// ---- POUs/HW/FB_EL2904_DiagnosticData.TcPOU
(****************************************************************************************)
(*							Beckhoff Automation Poland									*)
(*									30.01.2017											*)
(*			Blok funkcyjny pobierający informacje diagnostyczne z modułu EL2904			*)
(*			v2.5:																		*)
(*				- bReset, wErrorCount, ACT_Reset zmiana nazw pozostalych akcji			*)
(*				- usunieta zmienna sPath												*)
(*			v2.4:																		*)
(*				- obsluga bledu															*)
(*			v2.3:																		*)
(*				- dostosowano do rozbudowanej struktury									*)
(*			v1.2:																		*)
(*				- uruchamianie zboczem narastającym bExecute							*)	
(*______________________________________________________________________________________*)

FUNCTION_BLOCK FB_EL2904_DiagnosticData IMPLEMENTS I_ErrorHandling
VAR_INPUT
	sNetId						: T_AmsNetId;					(* Adres mastera EtherCAT *)
	uiSlaveAddr					: UINT;							(* Adres slave EtherCAT modułu EL2904 *)
	bExecute					: BOOL;							(* Zbocze narastające aktywuje komende *)
	bReset						: BOOL;							(* 	*)
END_VAR
VAR_OUTPUT
	stEL2904_DiagnosticData		: ST_EL2904_DiagnosticData;		(* Wyjściowa struktura danych *)
	bBusy						: BOOL;							(* Wyjście jest ustawione gdy aktualnie wykonywana jest komenda *)
	bError						: BOOL;							(* Wyjście jest ustawione gdy wystąpił błąd *) 
	udiErrorId					: UDINT;						(* Kod błedu *)
	bNewData					: BOOL;							(* Po otrzymaniu nowych danych przyjmuje wartość TRUE na jeden cykl *)
END_VAR
VAR
	fbEcCoESdoRead				: FB_EcCoESdoRead;
	stTempData					: ST_EL2904_DiagnosticData;		(* Tymczasowa struktura danych *)
	BSubIndex					: BYTE;
	wIndex						: WORD;
	iStep						: INT;
	pDstBuf						: PVOID;
	cbBufLen					: UDINT;
	rtExecute					: R_TRIG;
	rtError						: R_TRIG;
	rtReset						: R_TRIG;
	bRead						: BOOL;							(* Odczyt *)
	wTemp_800E_0C				: WORD;							(* Wartosc tymczasowa *)
	wTemp_800E_0D				: WORD;							(* Wartosc tymczasowa *)
	wTemp_800E_0E				: WORD;							(* Wartosc tymczasowa *)
	wErrorCount					: WORD;							// Licznik bledow
END_VAR

ACT_Reset(); 									// Wywolanie akcji resetu

rtExecute(CLK:=bExecute);

CASE iStep OF		
	(* Wspolne *)	
	0:												(* Odczyt nazwy modułu *)
		bNewData	:= FALSE;
		bRead		:= FALSE;
		IF rtExecute.Q THEN
			bBusy			:= TRUE;
			bError			:= FALSE;
			udiErrorId		:= 0;
			wIndex 			:= 16#1008;
			BSubIndex 		:= 0;
			pDstBuf 		:= ADR (stTempData.sDeviceName);
			cbBufLen 		:= SIZEOF(stTempData.sDeviceName);
			bRead			:= TRUE;
			iStep			:= iStep + 10;
		END_IF
	10:												(* Odczyt wersji HW *)
		bRead		:= FALSE;
		IF NOT fbEcCoESdoRead.bBusy AND NOT fbEcCoESdoRead.bError THEN
			wIndex 			:= 16#1009;
			BSubIndex 		:= 0;
			pDstBuf 		:= ADR (stTempData.sHardwareVersion);
			cbBufLen 		:= SIZEOF(stTempData.sHardwareVersion);
			bRead			:= TRUE;
			iStep			:= iStep + 10;
		END_IF
	20:												(* Odczyt wersji SW *)
		bRead				:= FALSE;
		IF NOT fbEcCoESdoRead.bBusy AND NOT fbEcCoESdoRead.bError THEN
			wIndex 			:= 16#100A;
			BSubIndex 		:= 0;
			pDstBuf 		:= ADR (stTempData.sSoftwareVersion);
			cbBufLen 		:= SIZEOF(stTempData.sSoftwareVersion);
			bRead			:= TRUE;
			iStep			:= iStep + 10;
		END_IF
	30:												(* Odczyt adresu FSoE *)
		bRead				:= FALSE;
		IF NOT fbEcCoESdoRead.bBusy AND NOT fbEcCoESdoRead.bError THEN
			wIndex 			:= 16#F980;
			BSubIndex 		:= 1;
			pDstBuf 		:= ADR (stTempData.dwFSoEAddress);
			cbBufLen 		:= SIZEOF(stTempData.dwFSoEAddress);
			bRead			:= TRUE;
			iStep			:= iStep + 10;
		END_IF;
	40:												(* Odczyt numeru seryjnego *)
		bRead				:= FALSE;
		IF NOT fbEcCoESdoRead.bBusy AND NOT fbEcCoESdoRead.bError THEN
			wIndex 			:= 16#F980;
			BSubIndex 		:= 2;
			pDstBuf 		:= ADR (stTempData.dwSerialNumber);
			cbBufLen 		:= SIZEOF(stTempData.dwSerialNumber);
			bRead			:= TRUE;
			iStep			:= iStep + 10;
		END_IF
	50:												(* Odczyt Temperature measurement 1 *)
		bRead				:= FALSE;
		IF NOT fbEcCoESdoRead.bBusy AND NOT fbEcCoESdoRead.bError THEN
			wIndex 			:= 16#FA80;
			BSubIndex 		:= 1;
			pDstBuf 		:= ADR (stTempData.wTemperaturePrimaryMC);
			cbBufLen 		:= SIZEOF(stTempData.wTemperaturePrimaryMC);
			bRead			:= TRUE;
			iStep			:= iStep + 10;
		END_IF
	60:												(* Odczyt Temperature measurement 2 *)
		bRead				:= FALSE;
		IF NOT fbEcCoESdoRead.bBusy AND NOT fbEcCoESdoRead.bError THEN
			wIndex 			:= 16#FA80;
			BSubIndex 		:= 2;
			pDstBuf 		:= ADR (stTempData.wTemperatureSecondaryMC);
			cbBufLen 		:= SIZEOF(stTempData.wTemperatureSecondaryMC);
			bRead			:= TRUE;
			iStep			:= iStep + 10;
		END_IF
	(*Charakterystyczne dla modulu *)
	70:												(* Odczyt FA80:03 Temperature Outputs *)
		bRead				:= FALSE;
		IF NOT fbEcCoESdoRead.bBusy AND NOT fbEcCoESdoRead.bError THEN
			wIndex 			:= 16#FA80;
			BSubIndex 		:= 3;
			pDstBuf 		:= ADR (stTempData.wTemperatureOut);
			cbBufLen 		:= SIZEOF(stTempData.wTemperatureOut);
			bRead			:= TRUE;
			iStep			:= iStep + 10;
		END_IF
	80:												(* Odczyt DO 1 *)
		bRead				:= FALSE;
		IF NOT fbEcCoESdoRead.bBusy AND NOT fbEcCoESdoRead.bError THEN
			wIndex 			:= 16#7001;
			BSubIndex 		:= 1;
			pDstBuf 		:= ADR(stTempData.bOutput1);
			cbBufLen 		:= SIZEOF(stTempData.bOutput1);
			bRead			:= TRUE;
			iStep			:= iStep + 10;
		END_IF
	90:												(* Odczyt DO 2 *)
		bRead				:= FALSE;
		IF NOT fbEcCoESdoRead.bBusy AND NOT fbEcCoESdoRead.bError THEN
			wIndex 			:= 16#7001;
			BSubIndex 		:= 2;
			pDstBuf 		:= ADR(stTempData.bOutput2);
			cbBufLen 		:= SIZEOF(stTempData.bOutput2);
			bRead			:= TRUE;
			iStep			:= iStep + 10;
		END_IF
	100:											(* Odczyt DO 3 *)
		bRead				:= FALSE;
		IF NOT fbEcCoESdoRead.bBusy AND NOT fbEcCoESdoRead.bError THEN
			wIndex 			:= 16#7001;
			BSubIndex 		:= 3;
			pDstBuf 		:= ADR(stTempData.bOutput3);
			cbBufLen 		:= SIZEOF(stTempData.bOutput3);
			bRead			:= TRUE;
			iStep			:= iStep + 10;
		END_IF
	110:											(* Odczyt DO 4 *)
		bRead				:= FALSE;
		IF NOT fbEcCoESdoRead.bBusy AND NOT fbEcCoESdoRead.bError THEN
			wIndex 			:= 16#7001;
			BSubIndex 		:= 4;
			pDstBuf 		:= ADR(stTempData.bOutput4);
			cbBufLen 		:= SIZEOF(stTempData.bOutput4);
			bRead			:= TRUE;
			iStep			:= iStep + 10;
		END_IF
	120:											(* Odczyt 800E 0C *)
		bRead				:= FALSE;
		IF NOT fbEcCoESdoRead.bBusy AND NOT fbEcCoESdoRead.bError THEN
			wIndex 			:= 16#800E;
			BSubIndex 		:= 16#0C;
			pDstBuf 		:= ADR (wTemp_800E_0C);
			cbBufLen 		:= SIZEOF(wTemp_800E_0C);
			bRead			:= TRUE;
			iStep			:= iStep + 10;
		END_IF
	130:											(* Odczyt 800E 0D *)
		bRead				:= FALSE;
		IF NOT fbEcCoESdoRead.bBusy AND NOT fbEcCoESdoRead.bError THEN
			wIndex 			:= 16#800E;
			BSubIndex 		:= 16#0D;
			pDstBuf 		:= ADR (wTemp_800E_0D);
			cbBufLen 		:= SIZEOF(wTemp_800E_0D);
			bRead			:= TRUE;
			iStep			:= iStep + 10;
		END_IF
	140:											(* Odczyt 800E 0E *)
		bRead				:= FALSE;
		IF NOT fbEcCoESdoRead.bBusy AND NOT fbEcCoESdoRead.bError THEN
			wIndex 			:= 16#800E;
			BSubIndex 		:= 16#0E;
			pDstBuf 		:= ADR (wTemp_800E_0E);
			cbBufLen 		:= SIZEOF(wTemp_800E_0E);
			bRead			:= TRUE;
			iStep			:= iStep + 10;
		END_IF
	
	150: (* Koniec odczytu *)
		bRead				:= FALSE;
		IF NOT fbEcCoESdoRead.bBusy AND NOT fbEcCoESdoRead.bError THEN
			iStep 			:= 200;
		END_IF
	200: (* Konwersje *)
		(* Zmiana numeru seryjnego na STRING *)
		stTempData.sSerialNumber 		:= '00000000';
		stTempData.sSerialNumber 		:= CONCAT(DELETE(stTempData.sSerialNumber, LEN(DWORD_TO_STRING(stTempData.dwSerialNumber)),1),DWORD_TO_STRING(stTempData.dwSerialNumber));
		stTempData.bOutputCross1 		:= wTemp_800E_0C.0;
		stTempData.bOutputCross2 		:= wTemp_800E_0C.1;
		stTempData.bOutputCross3 		:= wTemp_800E_0C.2;
		stTempData.bOutputCross4 		:= wTemp_800E_0C.3;
		stTempData.bOutputOpen1 		:= wTemp_800E_0C.4;
		stTempData.bOutputOpen2 		:= wTemp_800E_0C.5;
		stTempData.bOutputOpen3 		:= wTemp_800E_0C.6;
		stTempData.bOutputOpen4 		:= wTemp_800E_0C.7;
		stTempData.bFieldVoltH 			:= wTemp_800E_0D.0;
		stTempData.bFieldVoltL	 		:= wTemp_800E_0D.1;
		stTempData.bTHUC1			 	:= wTemp_800E_0E.0;
		stTempData.bTHUC2			 	:= wTemp_800E_0E.1;
		stTempData.bTOutBoardH		 	:= wTemp_800E_0E.2;
		stTempData.bTLUC1			 	:= wTemp_800E_0E.3;
		stTempData.bTLUC2			 	:= wTemp_800E_0E.4;
		stTempData.bTOutBoardL		 	:= wTemp_800E_0E.5;
		stTempData.bTDiffProcBoard	 	:= wTemp_800E_0E.6;
		stTempData.bTDiffBoards		 	:= wTemp_800E_0E.7;
		(* General Error bit *)
		stTempData.bGeneralError := stTempData.bOutputCross1 OR stTempData.bOutputCross2 OR stTempData.bOutputCross3 OR stTempData.bOutputCross4 OR
									stTempData.bOutputOpen1 OR stTempData.bOutputOpen2 OR stTempData.bOutputOpen3 OR stTempData.bOutputOpen4 OR
									stTempData.bFieldVoltH OR stTempData.bFieldVoltL OR stTempData.bTHUC1 OR stTempData.bTHUC2 OR stTempData.bTOutBoardH OR
									stTempData.bTLUC1 OR stTempData.bTLUC2 OR stTempData.bTOutBoardL OR stTempData.bTDiffProcBoard OR stTempData.bTDiffBoards;
		
		(* Przepisanie danych tymczasowych na wyjscie *)	
		stEL2904_DiagnosticData := stTempData;
		(* Ustawienie flag i powrot do poczatku *)
		bBusy							:= FALSE;
		bNewData						:= TRUE;
		iStep 							:= 0;
	1000: (* ERROR *)
		wErrorCount 					:= wErrorCount + 1;			// Inkrementacja licznika bledow
		iStep 							:= 0;
END_CASE

fbEcCoESdoRead(
	sNetId		:= sNetId,
	nSlaveAddr	:= uiSlaveAddr,
	nSubIndex	:= BSubIndex,
	nIndex		:= wIndex,
	pDstBuf		:= pDstBuf,
	cbBufLen	:= cbBufLen,
	bExecute 	:= bRead);
	
ACT_Error();

ACTION ACT_Error:
rtError(CLK:= fbEcCoESdoRead.bError, Q=> );
IF rtError.Q THEN
	bBusy 			:= FALSE;
	bError 			:= TRUE;
	bRead			:= FALSE;
	udiErrorId 		:= fbEcCoESdoRead.nErrId;
	iStep 			:= 1000;
END_IF
END_ACTION

ACTION ACT_Reset:
rtReset(CLK:= bReset, Q=> );			// Wywolanie triggera, wykrycie zbocza narastajacego zmiennej wejsciowej bReset
IF rtReset.Q THEN
	bBusy						:= FALSE;
	bError						:= FALSE;
	bNewData					:= FALSE;
	bRead						:= FALSE;
	iStep						:= 0;
	udiErrorId					:= 0;
END_IF
END_ACTION

PROPERTY P_Error : BOOL
GET
END_GET
END_PROPERTY

PROPERTY P_ErrorID : UDINT
GET
END_GET
END_PROPERTY

{attribute 'object_name' := 'ToString'}
METHOD ToString : STRING(255)
END_METHOD

END_FUNCTION_BLOCK

// ---- POUs/HW/FB_EL6900_DiagnosticData.TcPOU
(****************************************************************************************)
(*							Beckhoff Automation Poland									*)
(*									30.01.2017											*)
(*			Blok funkcyjny pobierający informacje diagnostyczne z modułu EL6900			*)
(*			v2.5:																		*)
(*				- bReset, wErrorCount, ACT_Reset zmiana nazw pozostalych akcji			*)
(*				- usunieta zmienna sPath												*)
(*			v2.4:																		*)
(*				- obsluga bledu															*)
(*			v2.3:																		*)
(*				- dostosowano do rozbudowanej struktury									*)
(*			v1.2:																		*)
(*				- uruchamianie zboczem narastającym bExecute							*)	
(*______________________________________________________________________________________*)

FUNCTION_BLOCK FB_EL6900_DiagnosticData IMPLEMENTS I_ErrorHandling
VAR_INPUT
	sNetId						: T_AmsNetId;					(* Adres mastera EtherCAT *)
	uiSlaveAddr					: UINT;							(* Adres slave EtherCAT modułu EL6900 *)
	bExecute					: BOOL;							(* Zbocze narastające aktywuje komende *)
	bReset						: BOOL;							(* 	*)
END_VAR
VAR_OUTPUT
	stEL6900_DiagnosticData		: ST_EL6900_DiagnosticData;		(* Wyjściowa struktura danych *)
	bBusy						: BOOL;							(* Wyjście jest ustawione gdy aktualnie wykonywana jest komenda *)
	bError						: BOOL;							(* Wyjście jest ustawione gdy wystąpił błąd *) 
	udiErrorId					: UDINT;						(* Kod błedu *)
	bNewData					: BOOL;							(* Po otrzymaniu nowych danych przyjmuje wartość TRUE na jeden cykl *)
END_VAR
VAR
	fbEcCoESdoRead				: FB_EcCoESdoRead;
	stTempData					: ST_EL6900_DiagnosticData;		(* Tymczasowa struktura danych *)
	BSubIndex					: BYTE;
	wIndex						: WORD;
	iStep						: INT;
	pDstBuf						: PVOID;
	cbBufLen					: UDINT;
	rtExecute					: R_TRIG;
	rtError						: R_TRIG;
	rtReset						: R_TRIG;
	bRead						: BOOL;							(* Odczyt *)
	wTemp_FA00_03				: WORD;							(* Wartosc tymczasowa *)
	wErrorCount					: WORD;							// Licznik bledow
END_VAR

ACT_Reset(); 									// Wywolanie akcji resetu

rtExecute(CLK:=bExecute);

CASE iStep OF		
	
	(* Wspolne *)	
	0:												(* Odczyt nazwy modułu *)
		bNewData	:= FALSE;
		bRead		:= FALSE;
		IF rtExecute.Q THEN
			bBusy			:= TRUE;
			bError			:= FALSE;
			udiErrorId		:= 0;
			wIndex 			:= 16#1008;
			BSubIndex 		:= 0;
			pDstBuf 		:= ADR (stTempData.sDeviceName);
			cbBufLen 		:= SIZEOF(stTempData.sDeviceName);
			bRead			:= TRUE;
			iStep			:= iStep + 10;
		END_IF
	10:												(* Odczyt wersji HW *)
		bRead		:= FALSE;
		IF NOT fbEcCoESdoRead.bBusy AND NOT fbEcCoESdoRead.bError THEN
			wIndex 			:= 16#1009;
			BSubIndex 		:= 0;
			pDstBuf 		:= ADR (stTempData.sHardwareVersion);
			cbBufLen 		:= SIZEOF(stTempData.sHardwareVersion);
			bRead			:= TRUE;
			iStep			:= iStep + 10;
		END_IF
	20:												(* Odczyt wersji SW *)
		bRead				:= FALSE;
		IF NOT fbEcCoESdoRead.bBusy AND NOT fbEcCoESdoRead.bError THEN
			wIndex 			:= 16#100A;
			BSubIndex 		:= 0;
			pDstBuf 		:= ADR (stTempData.sSoftwareVersion);
			cbBufLen 		:= SIZEOF(stTempData.sSoftwareVersion);
			bRead			:= TRUE;
			iStep			:= iStep + 10;
		END_IF
	30:												(* Odczyt adresu FSoE *)
		bRead				:= FALSE;
		IF NOT fbEcCoESdoRead.bBusy AND NOT fbEcCoESdoRead.bError THEN
			wIndex 			:= 16#F980;
			BSubIndex 		:= 1;
			pDstBuf 		:= ADR (stTempData.dwFSoEAddress);
			cbBufLen 		:= SIZEOF(stTempData.dwFSoEAddress);
			bRead			:= TRUE;
			iStep			:= iStep + 10;
		END_IF;
	40:												(* Odczyt numeru seryjnego *)
		bRead				:= FALSE;
		IF NOT fbEcCoESdoRead.bBusy AND NOT fbEcCoESdoRead.bError THEN
			wIndex 			:= 16#F980;
			BSubIndex 		:= 2;
			pDstBuf 		:= ADR (stTempData.dwSerialNumber);
			cbBufLen 		:= SIZEOF(stTempData.dwSerialNumber);
			bRead			:= TRUE;
			iStep			:= iStep + 10;
		END_IF
	50:												(* Odczyt Temperature measurement 1 *)
		bRead				:= FALSE;
		IF NOT fbEcCoESdoRead.bBusy AND NOT fbEcCoESdoRead.bError THEN
			wIndex 			:= 16#FA80;
			BSubIndex 		:= 1;
			pDstBuf 		:= ADR (stTempData.wTemperaturePrimaryMC);
			cbBufLen 		:= SIZEOF(stTempData.wTemperaturePrimaryMC);
			bRead			:= TRUE;
			iStep			:= iStep + 10;
		END_IF
	60:												(* Odczyt Temperature measurement 2 *)
		bRead				:= FALSE;
		IF NOT fbEcCoESdoRead.bBusy AND NOT fbEcCoESdoRead.bError THEN
			wIndex 			:= 16#FA80;
			BSubIndex 		:= 2;
			pDstBuf 		:= ADR (stTempData.wTemperatureSecondaryMC);
			cbBufLen 		:= SIZEOF(stTempData.wTemperatureSecondaryMC);
			bRead			:= TRUE;
			iStep			:= iStep + 10;
		END_IF
	(*Charakterystyczne dla modulu *)
	70:												(* Odczyt CRC projektu *)
		bRead				:= FALSE;
		IF NOT fbEcCoESdoRead.bBusy AND NOT fbEcCoESdoRead.bError THEN
			wIndex 			:= 16#F980;
			BSubIndex 		:= 3;
			pDstBuf 		:= ADR (stTempData.dwProjectCRC);
			cbBufLen 		:= SIZEOF(stTempData.dwProjectCRC);
			bRead			:= TRUE;
			iStep			:= iStep + 10;
		END_IF
	80:												(* Odczyt Safety Project State *)
		bRead				:= FALSE;
		IF NOT fbEcCoESdoRead.bBusy AND NOT fbEcCoESdoRead.bError THEN
			wIndex 			:= 16#F100;
			BSubIndex 		:= 1;
			pDstBuf 		:= ADR (stTempData.wSafetyProjectState);
			cbBufLen 		:= SIZEOF(stTempData.wSafetyProjectState);
			bRead			:= TRUE;
			iStep			:= iStep + 10;
		END_IF
	90:												(* Odczyt Vcc Primary MC*)
		bRead				:= FALSE;
		IF NOT fbEcCoESdoRead.bBusy AND NOT fbEcCoESdoRead.bError THEN
			wIndex 			:= 16#FA80;
			BSubIndex 		:= 3;
			pDstBuf 		:= ADR (stTempData.wVccPrimaryMC);
			cbBufLen 		:= SIZEOF(stTempData.wVccPrimaryMC);
			bRead			:= TRUE;
			iStep			:= iStep + 10;
		END_IF
	100:											(* Odczyt Vcc Secondary MC*)
		bRead				:= FALSE;
		IF NOT fbEcCoESdoRead.bBusy AND NOT fbEcCoESdoRead.bError THEN
			wIndex 			:= 16#FA80;
			BSubIndex 		:= 4;
			pDstBuf 		:= ADR (stTempData.wVccSecondaryMC);
			cbBufLen 		:= SIZEOF(stTempData.wVccSecondaryMC);
			bRead			:= TRUE;
			iStep			:= iStep + 10;
		END_IF
	110:											(* Odczyt FA00:03 Temperature error / Supply error *)
		bRead				:= FALSE;
		IF NOT fbEcCoESdoRead.bBusy AND NOT fbEcCoESdoRead.bError THEN
			wIndex 			:= 16#FA00;
			BSubIndex 		:= 3;
			pDstBuf 		:= ADR (wTemp_FA00_03);
			cbBufLen 		:= SIZEOF(wTemp_FA00_03);
			bRead			:= TRUE;
			iStep			:= iStep + 10;
		END_IF
	120: (* Koniec odczytu *)
		bRead				:= FALSE;
		IF NOT fbEcCoESdoRead.bBusy AND NOT fbEcCoESdoRead.bError THEN
			iStep 			:= 200;
		END_IF
	200: (* Konwersje *)
		(* Zmiana numeru seryjnego na STRING *)
		stTempData.sSerialNumber 		:= '00000000';
		stTempData.sSerialNumber 		:= CONCAT(DELETE(stTempData.sSerialNumber, LEN(DWORD_TO_STRING(stTempData.dwSerialNumber)),1),DWORD_TO_STRING(stTempData.dwSerialNumber));
		(* Zmiana CRC na STRING *)
		stTempData.sProjectCRC 			:= F_SAFETY_DWORD_TO_STIRNGHEX(stTempData.dwProjectCRC);
		(* Zmiana Project State na ENUM *)
		stTempData.eSAFETY_ProjectState	:= WORD_TO_INT(stTempData.wSafetyProjectState);
		(* Dekodowanie FA00:03 Temperature error / Supply error *)
		stTempData.bTempMax 			:= wTemp_FA00_03 = 16#0005;
		stTempData.bTempMin 			:= wTemp_FA00_03 = 16#0006;
		stTempData.bTempDiff 			:= wTemp_FA00_03 = 16#0007;
		stTempData.bSuppVoltuMaxC1		:= wTemp_FA00_03 = 16#0101;
		stTempData.bSuppVoltuMaxC2		:= wTemp_FA00_03 = 16#0102;
		stTempData.bSuppVoltuMinC1		:= wTemp_FA00_03 = 16#0103;
		stTempData.bSuppVoltuMinC2		:= wTemp_FA00_03 = 16#0104;
		(* General Error bit *)
		stTempData.bGeneralError := stTempData.bTempMax OR stTempData.bTempMin OR stTempData.bTempDiff OR
									stTempData.bSuppVoltuMaxC1 OR stTempData.bSuppVoltuMaxC2 OR stTempData.bSuppVoltuMinC1 OR stTempData.bSuppVoltuMinC2;
		(* Przepisanie danych tymczasowych na wyjscie *)	
		stEL6900_DiagnosticData 		:= stTempData;
		(* Ustawienie flag i powrot do poczatku *)
		bBusy							:= FALSE;
		bNewData						:= TRUE;
		iStep 							:= 0;
	1000: (* ERROR *)
		wErrorCount 					:= wErrorCount + 1;			// Inkrementacja licznika bledow
		iStep 							:= 0;
END_CASE

fbEcCoESdoRead(
	sNetId		:= sNetId,
	nSlaveAddr	:= uiSlaveAddr,
	nSubIndex	:= BSubIndex,
	nIndex		:= wIndex,
	pDstBuf		:= pDstBuf,
	cbBufLen	:= cbBufLen,
	bExecute 	:= bRead);
	
ACT_Error();

ACTION ACT_Error:
rtError(CLK:= fbEcCoESdoRead.bError, Q=> );
IF rtError.Q THEN
	bBusy 			:= FALSE;
	bError 			:= TRUE;
	bRead			:= FALSE;
	udiErrorId 		:= fbEcCoESdoRead.nErrId;
	iStep 			:= 1000;
END_IF
END_ACTION

ACTION ACT_Reset:
rtReset(CLK:= bReset, Q=> );			// Wywolanie triggera, wykrycie zbocza narastajacego zmiennej wejsciowej bReset
IF rtReset.Q THEN
	bBusy						:= FALSE;
	bError						:= FALSE;
	bNewData					:= FALSE;
	bRead						:= FALSE;
	iStep						:= 0;
	udiErrorId					:= 0;
END_IF
END_ACTION

PROPERTY P_Error : BOOL
GET
END_GET
END_PROPERTY

PROPERTY P_ErrorID : UDINT
GET
END_GET
END_PROPERTY

{attribute 'object_name' := 'ToString'}
METHOD ToString : STRING(255)
END_METHOD

END_FUNCTION_BLOCK

// ---- POUs/Others/F_SAFETY_DWORD_TO_STIRNGHEX.TcPOU
///*************************************************************************************************************************
///							Beckhoff Automation Poland									
///				`        	F_SAFETY_DWORD_TO_STIRNGHEX v1.0							
///									13.03.2015											
///				Funkcja zwraca napis zawierający zapis liczby w formacie szesnastkowym.			
///_______________________________________________________________________________________
FUNCTION F_SAFETY_DWORD_TO_STIRNGHEX : STRING(8)
VAR_INPUT
	dwIn: DWORD;
END_VAR
VAR
	dwTemp: DWORD;
	i: INT;
END_VAR

FOR i := 0 TO 7 DO
	dwTemp := ROR(dwIn,4*i) AND 16#F;

	CASE dwTemp OF
	0..9:
		F_SAFETY_DWORD_TO_STIRNGHEX := CONCAT(DWORD_TO_STRING(dwTemp), F_SAFETY_DWORD_TO_STIRNGHEX);
	10:
		F_SAFETY_DWORD_TO_STIRNGHEX := CONCAT('A', F_SAFETY_DWORD_TO_STIRNGHEX);
	11:
		F_SAFETY_DWORD_TO_STIRNGHEX := CONCAT('B', F_SAFETY_DWORD_TO_STIRNGHEX);
	12:
		F_SAFETY_DWORD_TO_STIRNGHEX := CONCAT('C', F_SAFETY_DWORD_TO_STIRNGHEX);
	13:
		F_SAFETY_DWORD_TO_STIRNGHEX := CONCAT('D', F_SAFETY_DWORD_TO_STIRNGHEX);
	14:
		F_SAFETY_DWORD_TO_STIRNGHEX := CONCAT('E', F_SAFETY_DWORD_TO_STIRNGHEX);
	15:
		F_SAFETY_DWORD_TO_STIRNGHEX := CONCAT('F', F_SAFETY_DWORD_TO_STIRNGHEX);
	END_CASE;
END_FOR
F_SAFETY_DWORD_TO_STIRNGHEX := DELETE(F_SAFETY_DWORD_TO_STIRNGHEX,4,1);

END_FUNCTION

// ---- POUs/HW/FB_EL6900_StatusData.TcPOU
(****************************************************************************************)
(*							Beckhoff Automation Poland									*)
(*									03.03.2017											*)
(*				Blok funkcyjny pobierający informacje diagnostyczne						*)
(*			 o blokach funkcyjnych, grupach, polaczeniach z modułu EL6900				*)
(*			V2.6:																		*)
(*				- Poprawiono bugi pętli FOR odczytu w akcjach ACT_StatusConnections		*)
(*					ACT_StatusFunctionBlocks i ACT_StatusGroups							*)
(*			v2.5:																		*)
(*				- bReset, wErrorCount, ACT_Reset zmiana nazw pozostalych akcji			*)
(*				- usunieta zmienna sPath												*)
(*			v2.4:																		*)
(*				- obsluga bledu															*)
(*			v2.3:																		*)
(*				- dostosowano do rozbudowanej struktury									*)
(*			v1.2:																		*)
(*				- uruchamianie zboczem narastającym bExecute							*)	
(*______________________________________________________________________________________*)

FUNCTION_BLOCK FB_EL6900_StatusData IMPLEMENTS I_ErrorHandling
VAR_INPUT
	sNetId						: T_AmsNetId;					(* Adres mastera EtherCAT *)
	uiSlaveAddr					: UINT;							(* Adres slave EtherCAT modułu EL6900 *)
	bExecute					: BOOL;							(* Zbocze narastające aktywuje komende *)
	bReset						: BOOL;							(* 	*)
END_VAR
VAR_OUTPUT
	stEL6900_StatusData			: ST_EL6900_StatusData;			(* Wyjściowa struktura danych *)
	bBusy						: BOOL;							(* Wyjście jest ustawione gdy aktualnie wykonywana jest komenda *)
	bError						: BOOL;							(* Wyjście jest ustawione gdy wystąpił błąd *) 
	udiErrorId					: UDINT;						(* Kod błedu *)
	bNewData					: BOOL;							(* Po otrzymaniu nowych danych przyjmuje wartość TRUE na jeden cykl *)
END_VAR
VAR
	fbEcCoESdoRead				: FB_EcCoESdoRead;
	BSubIndex					: BYTE;
	wIndex						: WORD;
	iInit						: INT:=10;
	pDstBuf						: PVOID;
	cbBufLen					: UDINT;
	ftRead						: F_TRIG;
	udiLastErrorID				: UDINT;
	tonRead						: TON;
	iStep						: INT:=0;
	BStatusConnections			: BYTE:=0;
	dwTempStatusConnection		: DWORD;						(* Wartosc tymczasowa *)
	BStatusGroups				: BYTE:=0;
	dwTempStatusGroups			: DWORD;						(* Wartosc tymczasowa *)
	BStatusFunctionBlocks		: BYTE:= 0;
	stEL6900_StatusData_Temp	: ST_EL6900_StatusData;			(* Wartosc tymczasowa *)
	index						: INT;
	bRead						: BOOL;
	rtExecute					: R_TRIG;
	rtError						: R_TRIG;
	rtReset						: R_TRIG;
	wErrorCount					: WORD;							// Licznik bledow
END_VAR

ACT_Reset(); 									// Wywolanie akcji resetu

rtExecute(CLK:=bExecute);
CASE iStep OF
	0:
		ACT_Init();
	10:
		bNewData:=FALSE;
		IF rtExecute.Q THEN
			iStep:=20;
			bBusy:=TRUE;
			bError:=FALSE;
			udiErrorId:=0;
		END_IF
	20:
		ACT_StatusConnections();

	30:
		ACT_StatusGroups();

	40:
		ACT_StatusFunctionBlocks();
	50:
		stEL6900_StatusData := stEL6900_StatusData_Temp;
		iStep:=10;
		bBusy:=FALSE;
		bNewData:=TRUE;
		bRead:=FALSE;
	1000:
		wErrorCount 					:= wErrorCount + 1;			// Inkrementacja licznika bledow
		iStep 							:= 0;
END_CASE

fbEcCoESdoRead(
	sNetId		:= sNetId,
	nSlaveAddr	:= uiSlaveAddr,
	nSubIndex	:= BSubIndex,
	nIndex		:= wIndex,
	pDstBuf		:= pDstBuf,
	cbBufLen	:= cbBufLen,
	bExecute 	:= bRead);
	
ACT_Error();

ACTION ACT_Error:
rtError(CLK:= fbEcCoESdoRead.bError, Q=> );
IF rtError.Q THEN
	bBusy 			:= FALSE;
	bError 			:= TRUE;
	bRead			:= FALSE;
	udiErrorId 		:= fbEcCoESdoRead.nErrId;
	iStep 			:= 1000;
END_IF
END_ACTION

ACTION ACT_Init:
CASE iInit OF
10:
	bRead:=FALSE;
	IF rtExecute.Q THEN
		bBusy:=TRUE;
		bError:=FALSE;
		udiErrorId:=0;
		bNewData:=FALSE;
		wIndex 			:= 16#2110;
		BSubIndex 		:= 0;
		pDstBuf 		:= ADR(stEL6900_StatusData_Temp.dwStatusConnections);
		cbBufLen 		:= SIZEOF(stEL6900_StatusData_Temp.dwStatusConnections);
		iInit:=iInit+10;
		bRead:=TRUE;
	END_IF
20:
	bRead:=FALSE;
	IF NOT fbEcCoESdoRead.bError AND NOT fbEcCoESdoRead.bBusy THEN
		wIndex 			:= 16#2120;
		BSubIndex 		:= 0;
		pDstBuf 		:= ADR(stEL6900_StatusData_Temp.dwStatusGroups);
		cbBufLen 		:= SIZEOF(stEL6900_StatusData_Temp.dwStatusGroups);
		iInit:=iInit+10;
		bRead:=TRUE;
	END_IF
30:
	bRead:=FALSE;
	IF NOT fbEcCoESdoRead.bError AND NOT fbEcCoESdoRead.bBusy THEN
		wIndex 			:= 16#2130;
		BSubIndex 		:= 0;
		pDstBuf 		:= ADR(stEL6900_StatusData_Temp.dwStatusFunctionBlocks);
		cbBufLen 		:= SIZEOF(stEL6900_StatusData_Temp.dwStatusFunctionBlocks);
		iInit:=iInit+10;
		bRead:=TRUE;
	END_IF
ELSE
	bRead:=FALSE;
	iInit:=10;
	iStep:=20;
END_CASE
END_ACTION

ACTION ACT_Reset:
rtReset(CLK:= bReset, Q=> );			// Wywolanie triggera, wykrycie zbocza narastajacego zmiennej wejsciowej bReset
IF rtReset.Q THEN
	bBusy						:= FALSE;
	bError						:= FALSE;
	bNewData					:= FALSE;
	bRead						:= FALSE;
	iStep						:= 0;
	udiErrorId					:= 0;
END_IF
END_ACTION

ACTION ACT_StatusConnections:
bRead:=FALSE;
IF NOT fbEcCoESdoRead.bError AND NOT fbEcCoESdoRead.bBusy THEN
	BStatusConnections := BStatusConnections + 1;
	IF bStatusConnections>1 THEN
		stEL6900_StatusData_Temp.arrstStatusConnections[BStatusConnections-1].dwStatusConnection := (dwTempStatusConnection);
		stEL6900_StatusData_Temp.arrstStatusConnections[BStatusConnections-1].BState:= DWORD_TO_BYTE(dwTempStatusConnection AND 16#000000FF);(*1B*)
		stEL6900_StatusData_Temp.arrstStatusConnections[BStatusConnections-1].BDiagnosis := DWORD_TO_BYTE(ROR(dwTempStatusConnection AND 16#0000FF00,8));(*2B*)
		stEL6900_StatusData_Temp.arrstStatusConnections[BStatusConnections-1].eSAFETY_ConnectionState:= stEL6900_StatusData_Temp.arrstStatusConnections[BStatusConnections-1].BState;
		stEL6900_StatusData_Temp.arrstStatusConnections[BStatusConnections-1].eSAFETY_ConnectionDiag0F := stEL6900_StatusData_Temp.arrstStatusConnections[BStatusConnections-1].BDiagnosis AND 16#0F;
		stEL6900_StatusData_Temp.arrstStatusConnections[BStatusConnections-1].BSAFETY_ConnectionDiagF0 := stEL6900_StatusData_Temp.arrstStatusConnections[BStatusConnections-1].BDiagnosis AND 16#F0;
		stEL6900_StatusData_Temp.arrstStatusConnections[BStatusConnections-1].sSAFETY_ConnectionDiagF0 := BYTE_TO_BINSTR(SHR(stEL6900_StatusData_Temp.arrstStatusConnections[BStatusConnections-1].BDiagnosis,4),4);
	END_IF
	IF BStatusConnections > stEL6900_StatusData_Temp.dwStatusConnections THEN
		BStatusConnections := 0;
		iStep := iStep + 10;
		bRead:=FALSE;
	ELSE
		wIndex 			:= 16#2110;
		BSubIndex 		:= 0+BStatusConnections;
		pDstBuf 		:= ADR(dwTempStatusConnection);
		cbBufLen 		:= SIZEOF(dwTempStatusConnection);
		bRead:=TRUE;
	END_IF
END_IF
END_ACTION

ACTION ACT_StatusFunctionBlocks:
bRead:=FALSE;
IF NOT fbEcCoESdoRead.bError AND NOT fbEcCoESdoRead.bBusy THEN
	BStatusFunctionBlocks := BStatusFunctionBlocks + 1;
	IF BStatusFunctionBlocks > stEL6900_StatusData_Temp.dwStatusFunctionBlocks THEN
		bRead:=FALSE;
		BStatusFunctionBlocks := 0;
		iStep := 50;
	ELSE
		wIndex 			:= 16#2130;
		BSubIndex 		:= BStatusFunctionBlocks;
		pDstBuf 		:= ADR(stEL6900_StatusData_Temp.arrstStatusFunctionBlocks[BStatusFunctionBlocks]);
		cbBufLen 		:= SIZEOF(stEL6900_StatusData_Temp.arrstStatusFunctionBlocks[BStatusFunctionBlocks]);
		bRead:=TRUE;
	END_IF
END_IF
END_ACTION

ACTION ACT_StatusGroups:
bRead:=FALSE;
IF NOT fbEcCoESdoRead.bError AND NOT fbEcCoESdoRead.bBusy THEN
	BStatusGroups := BStatusGroups + 1;	
	IF BStatusGroups>1 THEN
		stEL6900_StatusData_Temp.arrstStatusGroups[BStatusGroups-1].dwStatusGroup := dwTempStatusGroups;
		stEL6900_StatusData_Temp.arrstStatusGroups[BStatusGroups-1].BState := DWORD_TO_BYTE(dwTempStatusGroups AND 16#000000FF);
		stEL6900_StatusData_Temp.arrstStatusGroups[BStatusGroups-1].eSAFETY_GroupState := stEL6900_StatusData_Temp.arrstStatusGroups[BStatusGroups-1].BState;
		stEL6900_StatusData_Temp.arrstStatusGroups[BStatusGroups-1].BDiagnosis := DWORD_TO_BYTE(ROR(dwTempStatusGroups AND 16#0000FF00,8));(*2B*)
		stEL6900_StatusData_Temp.arrstStatusGroups[BStatusGroups-1].BInputs := DWORD_TO_BYTE(ROR(dwTempStatusGroups AND 16#00FF0000,16));(*3B*)
		stEL6900_StatusData_Temp.arrstStatusGroups[BStatusGroups-1].BOutputs := DWORD_TO_BYTE(ROR(dwTempStatusGroups AND 16#FF000000,24));(*4B*)
		stEL6900_StatusData_Temp.arrstStatusGroups[BStatusGroups-1].bRUN_STOP := stEL6900_StatusData_Temp.arrstStatusGroups[BStatusGroups-1].BInputs.0;
		stEL6900_StatusData_Temp.arrstStatusGroups[BStatusGroups-1].bERR_Ack := stEL6900_StatusData_Temp.arrstStatusGroups[BStatusGroups-1].BInputs.1;
		stEL6900_StatusData_Temp.arrstStatusGroups[BStatusGroups-1].bFB_ERR := stEL6900_StatusData_Temp.arrstStatusGroups[BStatusGroups-1].BOutputs.0;
		stEL6900_StatusData_Temp.arrstStatusGroups[BStatusGroups-1].bCOM_ERR := stEL6900_StatusData_Temp.arrstStatusGroups[BStatusGroups-1].BOutputs.1;
		stEL6900_StatusData_Temp.arrstStatusGroups[BStatusGroups-1].bOUT_ERR := stEL6900_StatusData_Temp.arrstStatusGroups[BStatusGroups-1].BOutputs.2;
	END_IF
	IF BStatusGroups > stEL6900_StatusData_Temp.dwStatusGroups THEN
		BStatusGroups := 0;
		iStep := iStep + 10;
		bRead:=FALSE;
	ELSE
		wIndex 			:= 16#2120;
		BSubIndex 		:= BStatusGroups;
		pDstBuf 		:= ADR(dwTempStatusGroups);
		cbBufLen 		:= SIZEOF(dwTempStatusGroups);
		bRead:=TRUE;
	END_IF
END_IF
END_ACTION

PROPERTY P_Error : BOOL
GET
END_GET
END_PROPERTY

PROPERTY P_ErrorID : UDINT
GET
END_GET
END_PROPERTY

{attribute 'object_name' := 'ToString'}
METHOD ToString : STRING(255)
END_METHOD

END_FUNCTION_BLOCK

// ---- POUs/FBs/F_SAFETY_StatusFB_TO_AND.TcPOU
FUNCTION F_SAFETY_StatusFB_TO_AND 	: ST_SAFETY_FBAND 		(* Struktura dedykowana *)
VAR_INPUT
	stFBStatus						: ST_SAFETY_FBStatus; 	(* Struktura ogolna *)
END_VAR

F_SAFETY_StatusFB_TO_AND.uStatus.stStatusWords 		:= stFBStatus;									(* Przepisanie *)
F_SAFETY_StatusFB_TO_AND.eState					 	:= stFBStatus.BState;							(* Ustawienie enum *)

END_FUNCTION

// ---- POUs/FBs/F_SAFETY_StatusFB_TO_CONNECTIONSHUTDOWN.TcPOU
FUNCTION F_SAFETY_StatusFB_TO_CONNECTIONSHUTDOWN : ST_SAFETY_FBCONNECTIONSHUTDOWN
VAR_INPUT
	stFBStatus						: ST_SAFETY_FBStatus; 	(* Struktura ogolna *)
END_VAR

F_SAFETY_StatusFB_TO_CONNECTIONSHUTDOWN.uStatus.stStatusWords	:= stFBStatus;									(* Przepisanie *)
F_SAFETY_StatusFB_TO_CONNECTIONSHUTDOWN.eState 					:= stFBStatus.BState;							(* Ustawienie enum *)
F_SAFETY_StatusFB_TO_CONNECTIONSHUTDOWN.bGeneralError			:= stFBStatus.wDiagnosis <> 0;					(* General Error *)

END_FUNCTION

// ---- POUs/FBs/F_SAFETY_StatusFB_TO_DECOUPLE.TcPOU
FUNCTION F_SAFETY_StatusFB_TO_DECOUPLE : ST_SAFETY_FBDECOUPLE
VAR_INPUT
	stFBStatus						: ST_SAFETY_FBStatus; 	(* Struktura ogolna *)
END_VAR

F_SAFETY_StatusFB_TO_DECOUPLE.uStatus.stStatusWords 		:= stFBStatus;					(* Przepisanie *)
F_SAFETY_StatusFB_TO_DECOUPLE.eState					 	:= stFBStatus.BState;			(* Ustawienie enum *)

END_FUNCTION

// ---- POUs/FBs/F_SAFETY_StatusFB_TO_EDM.TcPOU
FUNCTION F_SAFETY_StatusFB_TO_EDM : ST_SAFETY_FBEDM
VAR_INPUT
	stFBStatus						: ST_SAFETY_FBStatus; 	(* Struktura ogolna *)
END_VAR

F_SAFETY_StatusFB_TO_EDM.uStatus.stStatusWords	:= stFBStatus;									(* Przepisanie *)
F_SAFETY_StatusFB_TO_EDM.eState 				:= stFBStatus.BState;							(* Ustawienie enum *)
F_SAFETY_StatusFB_TO_EDM.bGeneralError			:= stFBStatus.wDiagnosis <> 0;					(* General Error *)

END_FUNCTION

// ---- POUs/FBs/F_SAFETY_StatusFB_TO_ESTOP.TcPOU
FUNCTION F_SAFETY_StatusFB_TO_ESTOP : ST_SAFETY_FBESTOP 	(* Struktura dedykowana *)
VAR_INPUT
	stFBStatus						: ST_SAFETY_FBStatus; 	(* Struktura ogolna *)
END_VAR

F_SAFETY_StatusFB_TO_ESTOP.uStatus.stStatusWords	:= stFBStatus;									(* Przepisanie *)
F_SAFETY_StatusFB_TO_ESTOP.eState 					:= stFBStatus.BState;							(* Ustawienie enum *)
F_SAFETY_StatusFB_TO_ESTOP.bGeneralError			:= stFBStatus.wDiagnosis <> 0;					(* General Error *)

END_FUNCTION

// ---- POUs/FBs/F_SAFETY_StatusFB_TO_MON.TcPOU
FUNCTION F_SAFETY_StatusFB_TO_MON : ST_SAFETY_FBMON
VAR_INPUT
	stFBStatus						: ST_SAFETY_FBStatus; 	(* Struktura ogolna *)
END_VAR

F_SAFETY_StatusFB_TO_MON.uStatus.stStatusWords	:= stFBStatus;									(* Przepisanie *)
F_SAFETY_StatusFB_TO_MON.eState 				:= stFBStatus.BState;							(* Ustawienie enum *)
F_SAFETY_StatusFB_TO_MON.bGeneralError			:= stFBStatus.wDiagnosis <> 0;					(* General Error *)

END_FUNCTION

// ---- POUs/FBs/F_SAFETY_StatusFB_TO_MUTING.TcPOU
FUNCTION F_SAFETY_StatusFB_TO_MUTING : ST_SAFETY_FBMUTING
VAR_INPUT
	stFBStatus						: ST_SAFETY_FBStatus; 	(* Struktura ogolna *)
END_VAR

F_SAFETY_StatusFB_TO_MUTING.uStatus.stStatusWords	:= stFBStatus;									(* Przepisanie *)
F_SAFETY_StatusFB_TO_MUTING.eState 					:= stFBStatus.BState;							(* Ustawienie enum *)
F_SAFETY_StatusFB_TO_MUTING.bGeneralError			:= stFBStatus.wDiagnosis <> 0;					(* General Error *)

END_FUNCTION

// ---- POUs/FBs/F_SAFETY_StatusFB_TO_OPMODE.TcPOU
FUNCTION F_SAFETY_StatusFB_TO_OPMODE : ST_SAFETY_FBOPMODE
VAR_INPUT
	stFBStatus						: ST_SAFETY_FBStatus; 	(* Struktura ogolna *)
END_VAR

F_SAFETY_StatusFB_TO_OPMODE.uStatus.stStatusWords	:= stFBStatus;									(* Przepisanie *)
F_SAFETY_StatusFB_TO_OPMODE.eState 					:= stFBStatus.BState;							(* Ustawienie enum *)
F_SAFETY_StatusFB_TO_OPMODE.bGeneralError			:= stFBStatus.wDiagnosis <> 0;					(* General Error *)

END_FUNCTION

// ---- POUs/FBs/F_SAFETY_StatusFB_TO_OR.TcPOU
FUNCTION F_SAFETY_StatusFB_TO_OR : ST_SAFETY_FBOR
VAR_INPUT
	stFBStatus						: ST_SAFETY_FBStatus; 	(* Struktura ogolna *)
END_VAR

F_SAFETY_StatusFB_TO_OR.uStatus.stStatusWords 		:= stFBStatus;									(* Przepisanie *)
F_SAFETY_StatusFB_TO_OR.eState					 	:= stFBStatus.BState;							(* Ustawienie enum *)

END_FUNCTION

// ---- POUs/FBs/F_SAFETY_StatusFB_TO_RS.TcPOU
FUNCTION F_SAFETY_StatusFB_TO_RS : ST_SAFETY_FBRS
VAR_INPUT
	stFBStatus						: ST_SAFETY_FBStatus; 	(* Struktura ogolna *)
END_VAR

F_SAFETY_StatusFB_TO_RS.uStatus.stStatusWords 		:= stFBStatus;									(* Przepisanie *)
F_SAFETY_StatusFB_TO_RS.eState					 	:= stFBStatus.BState;							(* Ustawienie enum *)

END_FUNCTION

// ---- POUs/FBs/F_SAFETY_StatusFB_TO_SR.TcPOU
FUNCTION F_SAFETY_StatusFB_TO_SR : ST_SAFETY_FBSR
VAR_INPUT
	stFBStatus						: ST_SAFETY_FBStatus; 	(* Struktura ogolna *)
END_VAR

F_SAFETY_StatusFB_TO_SR.uStatus.stStatusWords 		:= stFBStatus;									(* Przepisanie *)
F_SAFETY_StatusFB_TO_SR.eState					 	:= stFBStatus.BState;							(* Ustawienie enum *)

END_FUNCTION

// ---- POUs/FBs/F_SAFETY_StatusFB_TO_TOF.TcPOU
FUNCTION F_SAFETY_StatusFB_TO_TOF : ST_SAFETY_FBTOF
VAR_INPUT
	stFBStatus						: ST_SAFETY_FBStatus; 	(* Struktura ogolna *)
END_VAR

F_SAFETY_StatusFB_TO_TOF.uStatus.stStatusWords 		:= stFBStatus;									(* Przepisanie *)
F_SAFETY_StatusFB_TO_TOF.eState					 	:= stFBStatus.BState;							(* Ustawienie enum *)

END_FUNCTION

// ---- POUs/FBs/F_SAFETY_StatusFB_TO_TON.TcPOU
FUNCTION F_SAFETY_StatusFB_TO_TON : ST_SAFETY_FBTON
VAR_INPUT
	stFBStatus						: ST_SAFETY_FBStatus; 	(* Struktura ogolna *)
END_VAR

F_SAFETY_StatusFB_TO_TON.uStatus.stStatusWords 		:= stFBStatus;									(* Przepisanie *)
F_SAFETY_StatusFB_TO_TON.eState					 	:= stFBStatus.BState;							(* Ustawienie enum *)

END_FUNCTION

// ---- POUs/FBs/F_SAFETY_StatusFB_TO_TWOHAND.TcPOU
FUNCTION F_SAFETY_StatusFB_TO_TWOHAND : ST_SAFETY_FBTWOHAND
VAR_INPUT
	stFBStatus						: ST_SAFETY_FBStatus; 	(* Struktura ogolna *)
END_VAR

F_SAFETY_StatusFB_TO_TWOHAND.uStatus.stStatusWords	:= stFBStatus;									(* Przepisanie *)
F_SAFETY_StatusFB_TO_TWOHAND.eState 					:= stFBStatus.BState;							(* Ustawienie enum *)
F_SAFETY_StatusFB_TO_TWOHAND.bGeneralError			:= stFBStatus.wDiagnosis <> 0;					(* General Error *)

END_FUNCTION

// ---- POUs/HW/FB_AX580x_DiagnosticData.TcPOU
(****************************************************************************************)
(*							Beckhoff Automation Poland									*)
(*									19.05.2017											*)
(*			Blok funkcyjny pobierający informacje diagnostyczne z modułu AX580x			*)
(*			v1.0:																		*)
(*				- First version based on EL1904 v2.4									*)
(*______________________________________________________________________________________*)

FUNCTION_BLOCK FB_AX580x_DiagnosticData IMPLEMENTS I_ErrorHandling
VAR_INPUT
	sNetId						: T_AmsNetId;					(* Adres master EtherCAT *)
	uiSlaveAddr					: UINT;							(* Adres slave EtherCAT modułu EL1904 *)
	bExecute					: BOOL;							(* Zbocze narastające aktywuje komende *)
END_VAR
VAR_OUTPUT
	stAX580x_DiagnosticData		: ST_AX580x_DiagnosticData;		(* Wyjściowa struktura danych *)
	bBusy						: BOOL;							(* Wyjście jest ustawione gdy aktualnie wykonywana jest komenda *)
	bError						: BOOL;							(* Wyjście jest ustawione gdy wystąpił błąd *) 
	udiErrorId					: UDINT;						(* Kod błedu *)
	bNewData					: BOOL;							(* Po otrzymaniu nowych danych przyjmuje wartość TRUE na jeden cykl *)
END_VAR
VAR
	fbEcCoESdoRead				: FB_EcCoESdoRead;
	stTempData					: ST_AX580x_DiagnosticData;		(* Tymczasowa struktura danych *)
	BSubIndex					: BYTE;
	wIndex						: WORD;
	iStep						: INT;
	pDstBuf						: PVOID;
	cbBufLen					: UDINT;
    sPath 						: STRING;
	rtExecute					: R_TRIG;
	rtError						: R_TRIG;
	bRead						: BOOL;							(* Odczyt *)
	wTemp_800E_0A				: WORD;							(* Wartosc tymczasowa *)
	wTemp_800E_0B				: WORD;							(* Wartosc tymczasowa *)
	wTemp_800E_0C				: WORD;							(* Wartosc tymczasowa *)
	wTemp_800E_0D				: WORD;							(* Wartosc tymczasowa *)
END_VAR

rtExecute(CLK:=bExecute);

CASE iStep OF	
	(* Wspolne *)	
	0:
												(* Read the module name *)
		bNewData	:= FALSE;
		bRead		:= FALSE;
		IF rtExecute.Q THEN
			bBusy			:= TRUE;
			bError			:= FALSE;
			udiErrorId		:= 0;
			wIndex 			:= 16#1008;
			BSubIndex 		:= 0;
			pDstBuf 		:= ADR (stTempData.sDeviceName);
			cbBufLen 		:= SIZEOF(stTempData.sDeviceName);
			bRead			:= TRUE;
			iStep			:= iStep + 10;
		END_IF
	10:												(* Read the HW version *)
		bRead		:= FALSE;
		IF NOT fbEcCoESdoRead.bBusy AND NOT fbEcCoESdoRead.bError THEN
			wIndex 			:= 16#1009;
			BSubIndex 		:= 0;
			pDstBuf 		:= ADR (stTempData.sHardwareVersion);
			cbBufLen 		:= SIZEOF(stTempData.sHardwareVersion);
			bRead			:= TRUE;
			iStep			:= iStep + 10;
		END_IF
	20:												(* Read the SW version *)
		bRead				:= FALSE;
		IF NOT fbEcCoESdoRead.bBusy AND NOT fbEcCoESdoRead.bError THEN
			wIndex 			:= 16#100A;
			BSubIndex 		:= 0;
			pDstBuf 		:= ADR (stTempData.sSoftwareVersion);
			cbBufLen 		:= SIZEOF(stTempData.sSoftwareVersion);
			bRead			:= TRUE;
			iStep			:= iStep + 10;
		END_IF
	30:												(* Read the FSoE address *)
		bRead				:= FALSE;
		IF NOT fbEcCoESdoRead.bBusy AND NOT fbEcCoESdoRead.bError THEN
			wIndex 			:= 16#F980;
			BSubIndex 		:= 1;
			pDstBuf 		:= ADR (stTempData.dwFSoEAddress);
			cbBufLen 		:= SIZEOF(stTempData.dwFSoEAddress);
			bRead			:= TRUE;
			iStep			:= iStep + 10;
		END_IF;
	40:												(* Read the serial no *)
		bRead				:= FALSE;
		IF NOT fbEcCoESdoRead.bBusy AND NOT fbEcCoESdoRead.bError THEN
			wIndex 			:= 16#F980;
			BSubIndex 		:= 2;
			pDstBuf 		:= ADR (stTempData.dwSerialNumber);
			cbBufLen 		:= SIZEOF(stTempData.dwSerialNumber);
			bRead			:= TRUE;
			iStep			:= iStep + 10;
		END_IF
	50:												(* Read temperature MC1 *)
		bRead				:= FALSE;
		IF NOT fbEcCoESdoRead.bBusy AND NOT fbEcCoESdoRead.bError THEN
			wIndex 			:= 16#FA80;
			BSubIndex 		:= 1;
			pDstBuf 		:= ADR (stTempData.wTemperaturePrimaryMC);
			cbBufLen 		:= SIZEOF(stTempData.wTemperaturePrimaryMC);
			bRead			:= TRUE;
			iStep			:= iStep + 10;
		END_IF
	60:												(* Read temperature MC2 *)
		bRead				:= FALSE;
		IF NOT fbEcCoESdoRead.bBusy AND NOT fbEcCoESdoRead.bError THEN
			wIndex 			:= 16#FA80;
			BSubIndex 		:= 2;
			pDstBuf 		:= ADR (stTempData.wTemperatureSecondaryMC);
			cbBufLen 		:= SIZEOF(stTempData.wTemperatureSecondaryMC);
			bRead			:= TRUE;
			iStep			:= iStep + 10;
		END_IF
	(* Module specific *)
	70:												(* Reason for switching off index 01 *)
		bRead				:= FALSE;
		IF NOT fbEcCoESdoRead.bBusy AND NOT fbEcCoESdoRead.bError THEN
			wIndex 			:= 16#FA82;
			BSubIndex 		:= 1;
			pDstBuf 		:= ADR(stTempData.CoE_0xFA82_01);
			cbBufLen 		:= SIZEOF(stTempData.CoE_0xFA82_01);
			bRead			:= TRUE;
			iStep			:= iStep + 10;
		END_IF
	80:												(* Reason for switching off index 02 *)
		bRead				:= FALSE;
		IF NOT fbEcCoESdoRead.bBusy AND NOT fbEcCoESdoRead.bError THEN
			wIndex 			:= 16#FA82;
			BSubIndex 		:= 2;
			pDstBuf 		:= ADR(stTempData.CoE_0xFA82_02);
			cbBufLen 		:= SIZEOF(stTempData.CoE_0xFA82_02);
			bRead			:= TRUE;
			iStep			:= iStep + 10;
		END_IF
	90:												(* Reason for switching off index 03 *)
		bRead				:= FALSE;
		IF NOT fbEcCoESdoRead.bBusy AND NOT fbEcCoESdoRead.bError THEN
			wIndex 			:= 16#FA82;
			BSubIndex 		:= 3;
			pDstBuf 		:= ADR(stTempData.CoE_0xFA82_03);
			cbBufLen 		:= SIZEOF(stTempData.CoE_0xFA82_03);
			bRead			:= TRUE;
			iStep			:= iStep + 10;
		END_IF
	100:											(* Reason for switching off index 04 *)
		bRead				:= FALSE;
		IF NOT fbEcCoESdoRead.bBusy AND NOT fbEcCoESdoRead.bError THEN
			wIndex 			:= 16#FA82;
			BSubIndex 		:= 4;
			pDstBuf 		:= ADR(stTempData.CoE_0xFA82_04);
			cbBufLen 		:= SIZEOF(stTempData.CoE_0xFA82_04);
			bRead			:= TRUE;
			iStep			:= iStep + 10;
		END_IF
	110:											(* Reason for shutdown index 01 *)
		bRead				:= FALSE;
		IF NOT fbEcCoESdoRead.bBusy AND NOT fbEcCoESdoRead.bError THEN
			wIndex 			:= 16#FA10;
			BSubIndex 		:= 1;
			pDstBuf 		:= ADR(stTempData.CoE_0xFA10_01);
			cbBufLen 		:= SIZEOF(stTempData.CoE_0xFA10_01);
			bRead			:= TRUE;
			iStep			:= iStep + 10;
		END_IF
	120:											(* Reason for shutdown index 02 *)
		bRead				:= FALSE;
		IF NOT fbEcCoESdoRead.bBusy AND NOT fbEcCoESdoRead.bError THEN
			wIndex 			:= 16#FA10;
			BSubIndex 		:= 2;
			pDstBuf 		:= ADR(stTempData.CoE_0xFA10_02);
			cbBufLen 		:= SIZEOF(stTempData.CoE_0xFA10_02);
			bRead			:= TRUE;
			iStep			:= iStep + 10;
		END_IF
	130:											(* Reason for shutdown index 03 *)
		bRead				:= FALSE;
		IF NOT fbEcCoESdoRead.bBusy AND NOT fbEcCoESdoRead.bError THEN
			wIndex 			:= 16#FA10;
			BSubIndex 		:= 3;
			pDstBuf 		:= ADR(stTempData.CoE_0xFA10_03);
			cbBufLen 		:= SIZEOF(stTempData.CoE_0xFA10_03);
			bRead			:= TRUE;
			iStep			:= iStep + 10;
		END_IF
	140:											(* Reason for shutdown index 04 *)
		bRead				:= FALSE;
		IF NOT fbEcCoESdoRead.bBusy AND NOT fbEcCoESdoRead.bError THEN
			wIndex 			:= 16#FA10;
			BSubIndex 		:= 4;
			pDstBuf 		:= ADR(stTempData.CoE_0xFA10_04);
			cbBufLen 		:= SIZEOF(stTempData.CoE_0xFA10_04);
			bRead			:= TRUE;
			iStep			:= iStep + 10;
		END_IF
	150:											(* Reason for shutdown index 05 *)
		bRead				:= FALSE;
		IF NOT fbEcCoESdoRead.bBusy AND NOT fbEcCoESdoRead.bError THEN
			wIndex 			:= 16#FA10;
			BSubIndex 		:= 5;
			pDstBuf 		:= ADR(stTempData.CoE_0xFA10_05);
			cbBufLen 		:= SIZEOF(stTempData.CoE_0xFA10_05);
			bRead			:= TRUE;
			iStep			:= iStep + 10;
		END_IF
	160:											(* Reason for shutdown index 06 *)
		bRead				:= FALSE;
		IF NOT fbEcCoESdoRead.bBusy AND NOT fbEcCoESdoRead.bError THEN
			wIndex 			:= 16#FA10;
			BSubIndex 		:= 6;
			pDstBuf 		:= ADR(stTempData.CoE_0xFA10_06);
			cbBufLen 		:= SIZEOF(stTempData.CoE_0xFA10_06);
			bRead			:= TRUE;
			iStep			:= iStep + 10;
		END_IF
	170:											(* Reason for shutdown index 07 *)
		bRead				:= FALSE;
		IF NOT fbEcCoESdoRead.bBusy AND NOT fbEcCoESdoRead.bError THEN
			wIndex 			:= 16#FA10;
			BSubIndex 		:= 7;
			pDstBuf 		:= ADR(stTempData.CoE_0xFA10_07);
			cbBufLen 		:= SIZEOF(stTempData.CoE_0xFA10_07);
			bRead			:= TRUE;
			iStep			:= iStep + 10;
		END_IF
	180:											(* Reason for shutdown index 08 *)
		bRead				:= FALSE;
		IF NOT fbEcCoESdoRead.bBusy AND NOT fbEcCoESdoRead.bError THEN
			wIndex 			:= 16#FA10;
			BSubIndex 		:= 8;
			pDstBuf 		:= ADR(stTempData.CoE_0xFA10_08);
			cbBufLen 		:= SIZEOF(stTempData.CoE_0xFA10_08);
			bRead			:= TRUE;
			iStep			:= iStep + 10;
		END_IF
	190: (* Koniec odczytu *)
		bRead				:= FALSE;
		IF NOT fbEcCoESdoRead.bBusy AND NOT fbEcCoESdoRead.bError THEN
			iStep 			:= 200;
		END_IF
	
	200: (* Konwersje *)
		(* Zmiana numeru seryjnego na STRING *)
		stTempData.sSerialNumber 		:= '00000000';
		stTempData.sSerialNumber 		:= CONCAT(DELETE(stTempData.sSerialNumber, LEN(DWORD_TO_STRING(stTempData.dwSerialNumber)),1),DWORD_TO_STRING(stTempData.dwSerialNumber));

		(* Collect axis errors *)
		stTempData.bAxis1_NoErrorReaction := FALSE;
		stTempData.bAxis1_STOErrorReaction := FALSE;
		stTempData.bAxis1_SS1ErrorReaction := FALSE;
		stTempData.bAxis2_NoErrorReaction := FALSE;
		stTempData.bAxis2_STOErrorReaction := FALSE;
		stTempData.bAxis2_SS1ErrorReaction := FALSE;
		stTempData.bError_FA10_xx := (stTempData.CoE_0xFA10_01 > 0 AND stTempData.CoE_0xFA10_01 < 9);// OR (stTempData.CoE_0xFA10_02 > 0) OR (stTempData.CoE_0xFA10_03 > 0) OR (stTempData.CoE_0xFA10_04 > 0) OR
									// (stTempData.CoE_0xFA10_05 > 0) OR (stTempData.CoE_0xFA10_06 > 0) OR (stTempData.CoE_0xFA10_07 > 0) OR (stTempData.CoE_0xFA10_08 > 0);
		// specific axis error
		IF stTempData.CoE_0xFA10_01 = 0 THEN 
			// axis 1
			IF stTempData.CoE_0xFA10_07 > 0 THEN	
				stTempData.bAxis1_STOErrorReaction := (stTempData.CoE_0xFA10_07 AND 16#FF) = 16#40;
				stTempData.bAxis1_SS1ErrorReaction := (stTempData.CoE_0xFA10_07 AND 16#FF) = 16#50;
			ELSE
				stTempData.bAxis1_NoErrorReaction := TRUE;
			END_IF
			// axis 2
			IF stTempData.CoE_0xFA10_08 > 0 THEN	
				stTempData.bAxis2_STOErrorReaction := (stTempData.CoE_0xFA10_08 AND 16#FF) = 16#40;
				stTempData.bAxis2_SS1ErrorReaction := (stTempData.CoE_0xFA10_08 AND 16#FF) = 16#50;
			ELSE
				stTempData.bAxis2_NoErrorReaction := TRUE;
			END_IF
		END_IF
		
		(* General Error bit *)
		stTempData.bGeneralError := stTempData.bError_FA10_xx OR stTempData.bAxis1_STOErrorReaction OR stTempData.bAxis1_SS1ErrorReaction OR stTempData.bAxis2_STOErrorReaction OR stTempData.bAxis2_SS1ErrorReaction;
		(* Przepisanie danych tymczasowych na wyjscie *)	
		stAX580x_DiagnosticData 		:= stTempData;
		(* Ustawienie flag i powrot do poczatku *)
		bBusy							:= FALSE;
		bNewData						:= TRUE;
		iStep 							:= 0;
		
	1000: (* ERROR *)
		iStep 							:= 0;
END_CASE

fbEcCoESdoRead(
	sNetId		:= sNetId,
	nSlaveAddr	:= uiSlaveAddr,
	nSubIndex	:= BSubIndex,
	nIndex		:= wIndex,
	pDstBuf		:= pDstBuf,
	cbBufLen	:= cbBufLen,
	bExecute 	:= bRead);
	
A_Error();

ACTION A_Error:
rtError(CLK:= fbEcCoESdoRead.bError, Q=> );
IF rtError.Q THEN
	bBusy 			:= FALSE;
	bError 			:= TRUE;
	bRead			:= FALSE;
	udiErrorId 		:= fbEcCoESdoRead.nErrId;
	iStep 			:= 1000;
END_IF
END_ACTION

PROPERTY P_Error : BOOL
GET
END_GET
END_PROPERTY

PROPERTY P_ErrorID : UDINT
GET
END_GET
END_PROPERTY

{attribute 'object_name' := 'ToString'}
METHOD ToString : STRING(255)
END_METHOD

END_FUNCTION_BLOCK

// ---- POUs/Others/F_SAFETY_DOUBLESWAPDWORD.TcPOU
///*********************************************************************************************
///							Beckhoff Automation Poland											
///				`        	F_SAFETY_DOUBLESWAPDWORD v1.0									
///									13.03.2015													
///				Funkcja przepisuje liczbę zamieniając kolejność bajtów - pierwszy staje się		
///									ostanim, drugi przedostatnim itd.								
///__________________________________________________________________________________
FUNCTION F_SAFETY_DOUBLESWAPDWORD : DWORD
VAR_INPUT
	dwIn: DWORD;
END_VAR

F_SAFETY_DOUBLESWAPDWORD := ROL(dwIn AND 16#0000_00FF,24)+ROL(dwIn AND 16#0000_FF00,8)+ROL(dwIn AND 16#00FF_0000,24)+ROL(dwIn AND 16#FF00_0000,8);

END_FUNCTION

// ---- Version/F_GetVersionSafetyDiag.TcPOU
(*************************************************************************************************)
(*							Beckhoff Automation Poland												*)
(*									24.05.2017														*)
(*	Biblioteka sluzaca do diagnozowania stanu modulow oraz blokow funkcyjnych SAFETY				*)	
(* 								v2.7																*)
(*	Dodano FB_AX580x_DiagnosticData	ST_AX580x_DiagnosticData										*)		
(* 								v2.6																*)
(*	FB_ELx9xx - dodano Resety, obsluge bledow, zunifikowano kod										*)	
(* 								v2.5																*)
(*	obsluga bledow w blokach EL, poprawiednie w wizualizacji wyswietlania nr seryjnego - wiodace 0	*)	
(* 								v2.4																*)
(*	dodano zborczy blad dla struktur - bGeneralError										 		*)
(* 								v2.3																*)
(*	dodano inf o dokumentacji, uzupelniono diagnostyke, rozbudowano struktury diagnostyczne HW 		*)	
(* 								v2.2																*)
(*	usunieto bitmapy																				*)
(* 																									*)
(*	poprzednie wersje - inf wew																		*)

	(* Based on docu:
						EL6900en v 2.0.0 Date 2016-03-17 
						EL1904en v 2.0.0 Date 2016-03-17 
						EL2904en v 2.0.1 Date 2016-04-24
		TC version: 4020.28
*)											
FUNCTION F_GetVersionSafetyDiag : UINT
VAR_INPUT
	nVersionElement: INT;
END_VAR

CASE nVersionElement OF
1:	(* major number *)
	F_GetVersionSafetyDiag := stLibVersion_TC3SafetyDiag.iMajor;
2:	(* minor number *)
	F_GetVersionSafetyDiag := stLibVersion_TC3SafetyDiag.iMinor;
3:	(* revision number *)
	F_GetVersionSafetyDiag := stLibVersion_TC3SafetyDiag.iRevision;
ELSE
	F_GetVersionSafetyDiag := 16#FFFF;
END_CASE

END_FUNCTION

// ---- GlobalTextList.TcGTLO
TEXTLIST GlobalTextList
  902 = '%s'
  968 = 'AND'
  967 = 'ANDIn1'
  609 = 'ANDIn2'
  606 = 'ANDIn3'
  607 = 'ANDIn4'
  610 = 'ANDIn5'
  608 = 'ANDIn6'
  965 = 'ANDIn7'
  611 = 'ANDIn8'
  966 = 'ANDOut'
  231 = 'COM_ERR'
  896 = 'CONNECTION %d'
  73 = 'ConnectionShutdown'
  74 = 'Deactivate1'
  75 = 'Deactivate2'
  909 = 'Deactivated'
  377 = 'DECIn1'
  382 = 'DECIn2'
  378 = 'DECIn3'
  383 = 'DECIn4'
  379 = 'DECIn5'
  381 = 'DECIn6'
  380 = 'DECIn7'
  384 = 'DECIn8'
  376 = 'DECOUPLE'
  385 = 'DECOut1'
  386 = 'DECOut2'
  387 = 'DECOut3'
  388 = 'DECOut4'
  212 = 'DECOut5'
  389 = 'DECOut6'
  213 = 'DECOut7'
  214 = 'DECOut8'
  827 = 'DErrorSIADE1_2'
  828 = 'DErrorSIADE3_4'
  829 = 'DErrorSIADE5_6'
  830 = 'DErrorSIADE7_8'
  950 = 'DeviceName: %s'
  907 = 'DIAG:'
  819 = 'DicsError3_4'
  217 = 'DiscErr1_2_3_4'
  910 = 'DiscErrCS1_2'
  9 = 'DiscError'
  992 = 'DiscError1_2'
  839 = 'DiscError3_4'
  820 = 'DiscError5_6'
  823 = 'DiscError7_8'
  840 = 'DiscErrorSec'
  1002 = 'DisErrorOSSD'
  679 = 'EDM'
  825 = 'EDM1'
  821 = 'EDM1Error'
  826 = 'EDM2'
  831 = 'EDM2Error'
  944 = 'EL1904 DIAGNOSTIC'
  1480 = 'EL2904 DIAGNOSTIC'
  461 = 'EL6900 DIAGNOSTIC'
  842 = 'EMD1Error'
  981 = 'EMD2'
  841 = 'EMD2Error'
  982 = 'Emergency Stop'
  980 = 'Enable'
  76 = 'Error'
  227 = 'ErrorAck'
  822 = 'EStopDelOut'
  991 = 'EStopIn1'
  990 = 'EStopIn2'
  984 = 'EStopIn3'
  985 = 'EStopIn4'
  986 = 'EStopIn5'
  987 = 'EStopIn6'
  988 = 'EStopIn7'
  989 = 'EStopIn8'
  824 = 'EStopOut'
  229 = 'FB_ERR'
  971 = 'FSoEAddress: %d'
  226 = 'GROUP %d'
  964 = 'HardwareVersion: %s'
  1019 = 'Input1'
  1012 = 'Input2'
  1005 = 'Input3'
  1006 = 'Input4'
  481 = 'MON'
  680 = 'MON1'
  681 = 'MON2'
  844 = 'MONDelOut'
  487 = 'MONIn1'
  486 = 'MONIn2'
  484 = 'MONIn3'
  482 = 'MONIn4'
  843 = 'MONOut'
  485 = 'MONSec1'
  483 = 'MONSec2'
  1001 = 'MuteDelOut'
  1000 = 'MuteOut'
  339 = 'MuteSeqViolated'
  998 = 'MUTING'
  979 = 'Muting1'
  993 = 'Muting2'
  994 = 'Muting3'
  996 = 'Muting4'
  999 = 'MutingActive'
  338 = 'MutingTimeEx'
  1530 = 'OpenCircuit1'
  1540 = 'OpenCircuit2'
  1293 = 'OpenCircuit3'
  1301 = 'OpenCircuit4'
  1 = 'OPIn1'
  2 = 'OPIn2'
  5 = 'OPIn3'
  4 = 'OPIn4'
  3 = 'OPIn5'
  8 = 'OPIn6'
  6 = 'OPIn7'
  7 = 'OPIn8'
  0 = 'OPMODE'
  12 = 'OPOut1'
  10 = 'OPOut2'
  11 = 'OPOut3'
  13 = 'OPOut4'
  16 = 'OPOut5'
  14 = 'OPOut6'
  895 = 'OPOut7'
  15 = 'OPOut8'
  327 = 'OR'
  330 = 'ORIn1'
  162 = 'ORIn2'
  333 = 'ORIn3'
  336 = 'ORIn4'
  340 = 'ORIn5'
  342 = 'ORIn6'
  345 = 'ORIn7'
  160 = 'ORIn8'
  163 = 'OROut'
  997 = 'OSSDIn1'
  995 = 'OSSDIn2'
  1490 = 'Output1'
  1500 = 'Output2'
  1510 = 'Output3'
  1520 = 'Output4'
  230 = 'OUT_ERR'
  464 = 'ProjectCRC: 0x%s'
  294 = 'Reset'
  983 = 'Restart'
  292 = 'RS'
  297 = 'RSOut'
  233 = 'RunStop'
  978 = 'SerialNumber: %s'
  299 = 'Set'
  957 = 'SoftwareVersion: %s'
  434 = 'SR'
  437 = 'SROut'
  913 = 'STATE:'
  682 = 'SwitchOffErr'
  683 = 'SwitchOnErr'
  1004 = 'TemperaturePrimaryMC: %d'
  1003 = 'TemperatureSecondaryMC: %d'
  1167 = 'TOF'
  1176 = 'TOFIn'
  1186 = 'TOFOut'
  270 = 'TON'
  272 = 'TONIn'
  274 = 'TONOut'
  204 = 'TWO HAND'
  216 = 'TwoHandErr'
  206 = 'TwoHandIn1'
  209 = 'TwoHandIn2'
  207 = 'TwoHandIn3'
  210 = 'TwoHandIn4'
  215 = 'TwoHandOut'
  205 = 'VccPrimaryMC: %d'
  208 = 'VccSecondaryMC: %d'
END_TEXTLIST

// ---- VISUs/FBs/TL_ConnectionDiag.TcTLO
TEXTLIST TL_ConnectionDiag
  0 = 'Without Errors'
  1 = 'Invalid Command'
  2 = 'Unknown Command'
  3 = 'Invalid Connection ID'
  4 = 'Invalid CRC'
  5 = 'Watchdog Time Elapsed'
  6 = 'Invalid FSo EAddress'
  7 = 'Invalid Data'
  8 = 'Invalid Comm Param Length'
  9 = 'Invalid Comm Params'
  10 = 'Invalid User Param Length'
  11 = 'Invalid User Params'
  12 = 'FSoE Master Reset\t'
  13 = 'Module Error'
  14 = 'EL290x Error'
  15 = 'Slave Not Yet Started'
   = ''
END_TEXTLIST

// ---- VISUs/FBs/TL_ConnectionState.TcTLO
TEXTLIST TL_ConnectionState
  0 = 'Unknown'
  100 = 'Reset'
  101 = 'Session'
  102 = 'Connection'
  103 = 'Parameter'
  104 = 'Data'
  105 = 'Shutdown'
   = ''
END_TEXTLIST

// ---- VISUs/FBs/TL_FbState.TcTLO
TEXTLIST TL_FbState
  0 = 'UNDEFINED'
  1 = 'RUN'
  2 = 'STOP'
  3 = 'SAFE'
  4 = 'ERROR'
  5 = 'RESET'
  6 = 'START'
  7 = 'ERROR DELAY'
  8 = 'DELAY OUT'
  9 = 'FUNC TEST'
  11 = '1 BUTTON'
  12 = '2 BUTTON'
  13 = 'REALISE'
  14 = 'MON OFF'
  15 = 'MON ON'
   = ''
END_TEXTLIST

// ---- VISUs/FBs/TL_FbStateCS.TcTLO
TEXTLIST TL_FbStateCS
  0 = 'UNDEFINED'
  1 = 'RUN'
  2 = 'STOP'
  3 = 'SAFE'
  4 = 'ERROR'
  5 = 'RESET'
  10 = 'ACTIVE'
  11 = 'DEACTIVE'
   = ''
END_TEXTLIST

// ---- VISUs/FBs/TL_FbStateMUTING.TcTLO
TEXTLIST TL_FbStateMUTING
  0 = 'UNDEFINED'
  1 = 'RUN'
  2 = 'STOP'
  3 = 'SAFE'
  4 = 'ERROR'
  5 = 'RESET'
  8 = 'DELAY OUT'
  9 = 'MUTING 1'
  10 = 'MUTING 2'
  11 = 'MUTING 3'
  12 = 'MUTING 4'
  13 = 'MUTING 5'
  14 = 'MUTING 6'
  15 = 'MUTING 7'
  16 = 'MUTING 8'
  17 = 'MUTING 9'
   = ''
END_TEXTLIST

// ---- VISUs/FBs/TL_FbStateSetReset.TcTLO
TEXTLIST TL_FbStateSetReset
  0 = 'UNDEFINED'
  2 = 'STOP'
  3 = 'SAFE'
  9 = 'SET'
   = ''
END_TEXTLIST

// ---- VISUs/FBs/TL_FbStateTimer.TcTLO
TEXTLIST TL_FbStateTimer
  0 = 'UNDEFINED'
  1 = 'RUN'
  2 = 'STOP'
  3 = 'SAFE'
  8 = 'DELAY OUT'
  9 = 'DELAY IN'
   = ''
END_TEXTLIST

// ---- VISUs/FBs/TL_GroupState.TcTLO
TEXTLIST TL_GroupState
  0 = 'UNKNOWN'
  1 = 'RUN'
  2 = 'STOP'
  3 = 'SAFE'
  4 = 'ERROR'
  5 = 'RESET'
   = ''
END_TEXTLIST

// ---- VISUs/FBs/V_PH_AND.TcVIS
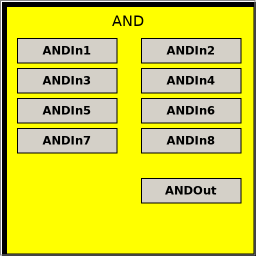
VISUALIZATION V_PH_AND  // 256x256
VAR_INPUT
	stSafetyAnd			:ST_SAFETY_FBAND;
END_VAR
    Rectangle (2,2 256x256), colour toggle: stSafetyAnd.bGeneralError
    RoundedRectangle (17,68 100x25), "ANDIn3", colour toggle: stSafetyAnd.uStatus.stStatusWords.wInputs.1
    RoundedRectangle (141,68 100x25), "ANDIn4", colour toggle: stSafetyAnd.uStatus.stStatusWords.wInputs.11
    RoundedRectangle (141,98 100x25), "ANDIn6", colour toggle: stSafetyAnd.uStatus.stStatusWords.wInputs.13
    RoundedRectangle (141,38 100x25), "ANDIn2", colour toggle: stSafetyAnd.uStatus.stStatusWords.wInputs.9
    RoundedRectangle (17,98 100x25), "ANDIn5", colour toggle: stSafetyAnd.uStatus.stStatusWords.wInputs.12
    RoundedRectangle (141,128 100x25), "ANDIn8", colour toggle: stSafetyAnd.uStatus.stStatusWords.wInputs.15
    RoundedRectangle (17,128 100x25), "ANDIn7", colour toggle: stSafetyAnd.uStatus.stStatusWords.wInputs.14
    RoundedRectangle (141,178 100x25), "ANDOut", colour toggle: stSafetyAnd.uStatus.stStatusWords.wOutputs.0
    RoundedRectangle (17,38 100x25), "ANDIn1", colour toggle: stSafetyAnd.uStatus.stStatusWords.wInputs.8
    Label (53,6 150x30), "AND"
    Textfield (17,226 234x25), text list: 'TL_FbState', text index: stSafetyAnd.eState
END_VISUALIZATION

// ---- VISUs/FBs/V_PH_CONNECTIONSHUTDOWN.TcVIS
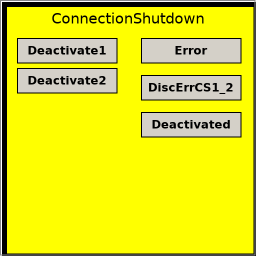
VISUALIZATION V_PH_CONNECTIONSHUTDOWN  // 256x256
VAR_INPUT
	stSafetyConnectionShutdown				:ST_SAFETY_FBCONNECTIONSHUTDOWN;
	
	
END_VAR
    Rectangle (2,2 256x256), colour toggle: stSafetyConnectionShutdown.bGeneralError
    Label (5,6 246x25), "ConnectionShutdown"
    RoundedRectangle (17,38 100x25), "Deactivate1", colour toggle: stSafetyConnectionShutdown.uStatus.stStatusWords.wInputs.8
    RoundedRectangle (17,68 100x25), "Deactivate2", colour toggle: stSafetyConnectionShutdown.uStatus.stStatusWords.wInputs.9
    RoundedRectangle (141,38 100x25), "Error", colour toggle: stSafetyConnectionShutdown.uStatus.stStatusWords.wOutputs.0
    RoundedRectangle (141,112 100x25), "Deactivated", colour toggle: stSafetyConnectionShutdown.uStatus.stStatusWords.wOutputs.1
    RoundedRectangle (141,75 100x25), "DiscErrCS1_2", colour toggle: stSafetyConnectionShutdown.uStatus.stStatusWords.wDiagnosis.0, invisible if: NOT stSafetyConnectionShutdown.uStatus.stStatusWords.wDiagnosis.0
    Textfield (17,226 234x25), text list: 'TL_FbStateCS', text index: stSafetyConnectionShutdown.eState
END_VISUALIZATION

// ---- VISUs/FBs/V_PH_DECOUPLE.TcVIS
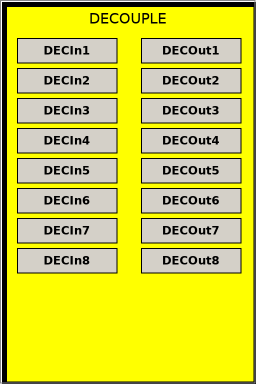
VISUALIZATION V_PH_DECOUPLE  // 256x384
VAR_INPUT
	stSafetyDecouple			: ST_SAFETY_FBDECOUPLE;
END_VAR
    Rectangle (2,2 256x384), colour toggle: stSafetyDecouple.bGeneralError
    Label (5,6 246x25), "DECOUPLE"
    RoundedRectangle (17,38 100x25), "DECIn1", colour toggle: stSafetyDecouple.uStatus.stStatusWords.wInputs.8
    RoundedRectangle (17,98 100x25), "DECIn3", colour toggle: stSafetyDecouple.uStatus.stStatusWords.wInputs.10
    RoundedRectangle (17,158 100x25), "DECIn5", colour toggle: stSafetyDecouple.uStatus.stStatusWords.wInputs.12
    RoundedRectangle (17,218 100x25), "DECIn7", colour toggle: stSafetyDecouple.uStatus.stStatusWords.wInputs.14
    RoundedRectangle (17,188 100x25), "DECIn6", colour toggle: stSafetyDecouple.uStatus.stStatusWords.wInputs.13
    RoundedRectangle (17,68 100x25), "DECIn2", colour toggle: stSafetyDecouple.uStatus.stStatusWords.wInputs.9
    RoundedRectangle (17,128 100x25), "DECIn4", colour toggle: stSafetyDecouple.uStatus.stStatusWords.wInputs.11
    RoundedRectangle (17,248 100x25), "DECIn8", colour toggle: stSafetyDecouple.uStatus.stStatusWords.wInputs.15
    RoundedRectangle (141,38 100x25), "DECOut1", colour toggle: stSafetyDecouple.uStatus.stStatusWords.wOutputs.8
    RoundedRectangle (141,68 100x25), "DECOut2", colour toggle: stSafetyDecouple.uStatus.stStatusWords.wOutputs.9
    RoundedRectangle (141,98 100x25), "DECOut3", colour toggle: stSafetyDecouple.uStatus.stStatusWords.wOutputs.10
    RoundedRectangle (141,128 100x25), "DECOut4", colour toggle: stSafetyDecouple.uStatus.stStatusWords.wOutputs.11
    RoundedRectangle (141,188 100x25), "DECOut6", colour toggle: stSafetyDecouple.uStatus.stStatusWords.wOutputs.13
    RoundedRectangle (141,158 100x25), "DECOut5", colour toggle: stSafetyDecouple.uStatus.stStatusWords.wOutputs.12
    RoundedRectangle (141,218 100x25), "DECOut7", colour toggle: stSafetyDecouple.uStatus.stStatusWords.wOutputs.14
    RoundedRectangle (141,248 100x25), "DECOut8", colour toggle: stSafetyDecouple.uStatus.stStatusWords.wOutputs.15
    Textfield (17,354 234x25), text list: 'TL_FbState', text index: stSafetyDecouple.eState
END_VISUALIZATION

// ---- VISUs/FBs/V_PH_EDM.TcVIS
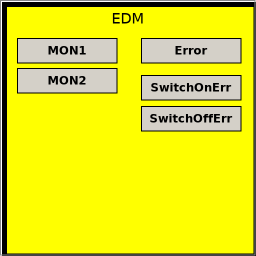
VISUALIZATION V_PH_EDM  // 256x256
VAR_INPUT
	stSafetyEDM				:ST_SAFETY_FBEDM;
	
	
END_VAR
    Rectangle (2,2 256x256), colour toggle: stSafetyEDM.bGeneralError
    Label (5,6 246x25), "EDM"
    RoundedRectangle (17,38 100x25), "MON1", colour toggle: stSafetyEDM.uStatus.stStatusWords.wInputs.8
    RoundedRectangle (141,38 100x25), "Error", colour toggle: stSafetyEDM.uStatus.stStatusWords.wOutputs.0
    RoundedRectangle (17,68 100x25), "MON2", colour toggle: stSafetyEDM.uStatus.stStatusWords.wInputs.9
    RoundedRectangle (141,106 100x25), "SwitchOffErr", colour toggle: stSafetyEDM.uStatus.stStatusWords.wDiagnosis.0, invisible if: NOT stSafetyEDM.uStatus.stStatusWords.wDiagnosis.0
    RoundedRectangle (141,75 100x25), "SwitchOnErr", colour toggle: stSafetyEDM.uStatus.stStatusWords.wDiagnosis.1, invisible if: NOT stSafetyEDM.uStatus.stStatusWords.wDiagnosis.1
    Textfield (17,226 234x25), text list: 'TL_FbState', text index: stSafetyEDM.eState
END_VISUALIZATION

// ---- VISUs/FBs/V_PH_ESTOP.TcVIS
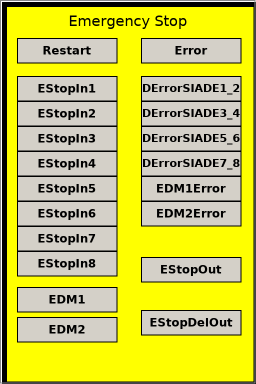
VISUALIZATION V_PH_ESTOP  // 256x384
VAR_INPUT
	stSafetyEStop				: ST_SAFETY_FBESTOP;
END_VAR
    Rectangle (2,2 256x384), colour toggle: stSafetyEStop.bGeneralError
    Label (53,6 150x30), "Emergency Stop"
    RoundedRectangle (17,38 100x25), "Restart", colour toggle: stSafetyEStop.uStatus.stStatusWords.wInputs.0
    RoundedRectangle (17,126 100x25), "EStopIn3", colour toggle: stSafetyEStop.uStatus.stStatusWords.wInputs.10
    RoundedRectangle (17,151 100x25), "EStopIn4", colour toggle: stSafetyEStop.uStatus.stStatusWords.wInputs.11
    RoundedRectangle (17,176 100x25), "EStopIn5", colour toggle: stSafetyEStop.uStatus.stStatusWords.wInputs.12
    RoundedRectangle (17,201 100x25), "EStopIn6", colour toggle: stSafetyEStop.uStatus.stStatusWords.wInputs.13
    RoundedRectangle (17,226 100x25), "EStopIn7", colour toggle: stSafetyEStop.uStatus.stStatusWords.wInputs.14
    RoundedRectangle (17,251 100x25), "EStopIn8", colour toggle: stSafetyEStop.uStatus.stStatusWords.wInputs.15
    RoundedRectangle (17,101 100x25), "EStopIn2", colour toggle: stSafetyEStop.uStatus.stStatusWords.wInputs.9
    RoundedRectangle (17,76 100x25), "EStopIn1", colour toggle: stSafetyEStop.uStatus.stStatusWords.wInputs.8
    RoundedRectangle (141,76 100x25), "DiscError1_2", colour toggle: stSafetyEStop.uStatus.stStatusWords.wDiagnosis.0, invisible if: NOT stSafetyEStop.uStatus.stStatusWords.wDiagnosis.0
    RoundedRectangle (141,101 100x25), "DicsError3_4", colour toggle: stSafetyEStop.uStatus.stStatusWords.wDiagnosis.1, invisible if: NOT stSafetyEStop.uStatus.stStatusWords.wDiagnosis.1
    RoundedRectangle (141,126 100x25), "DiscError5_6", colour toggle: stSafetyEStop.uStatus.stStatusWords.wDiagnosis.2, invisible if: NOT stSafetyEStop.uStatus.stStatusWords.wDiagnosis.2
    RoundedRectangle (141,176 100x25), "EDM1Error", colour toggle: stSafetyEStop.uStatus.stStatusWords.wDiagnosis.4, invisible if: NOT stSafetyEStop.uStatus.stStatusWords.wDiagnosis.4
    RoundedRectangle (141,310 100x25), "EStopDelOut", colour toggle: stSafetyEStop.uStatus.stStatusWords.wOutputs.2
    RoundedRectangle (141,38 100x25), "Error", colour toggle: stSafetyEStop.uStatus.stStatusWords.wOutputs.0
    RoundedRectangle (141,151 100x25), "DiscError7_8", colour toggle: stSafetyEStop.uStatus.stStatusWords.wDiagnosis.3, invisible if: NOT stSafetyEStop.uStatus.stStatusWords.wDiagnosis.3
    RoundedRectangle (141,257 100x25), "EStopOut", colour toggle: stSafetyEStop.uStatus.stStatusWords.wOutputs.1
    RoundedRectangle (17,287 100x25), "EDM1", colour toggle: stSafetyEStop.uStatus.stStatusWords.wInputs.1
    RoundedRectangle (17,317 100x25), "EDM2", colour toggle: stSafetyEStop.uStatus.stStatusWords.wInputs.2
    RoundedRectangle (141,76 100x25), "DErrorSIADE1_2", colour toggle: stSafetyEStop.uStatus.stStatusWords.wDiagnosis.8, invisible if: NOT stSafetyEStop.uStatus.stStatusWords.wDiagnosis.8
    RoundedRectangle (141,101 100x25), "DErrorSIADE3_4", colour toggle: stSafetyEStop.uStatus.stStatusWords.wDiagnosis.9, invisible if: NOT stSafetyEStop.uStatus.stStatusWords.wDiagnosis.9
    RoundedRectangle (141,126 100x25), "DErrorSIADE5_6", colour toggle: stSafetyEStop.uStatus.stStatusWords.wDiagnosis.10, invisible if: NOT stSafetyEStop.uStatus.stStatusWords.wDiagnosis.10
    RoundedRectangle (141,151 100x25), "DErrorSIADE7_8", colour toggle: stSafetyEStop.uStatus.stStatusWords.wDiagnosis.11, invisible if: NOT stSafetyEStop.uStatus.stStatusWords.wDiagnosis.11
    RoundedRectangle (141,201 100x25), "EDM2Error", colour toggle: stSafetyEStop.uStatus.stStatusWords.wDiagnosis.5, invisible if: NOT stSafetyEStop.uStatus.stStatusWords.wDiagnosis.5
    Textfield (17,354 234x25), text list: 'TL_FbState', text index: stSafetyEStop.eState
END_VISUALIZATION

// ---- VISUs/FBs/V_PH_MON.TcVIS
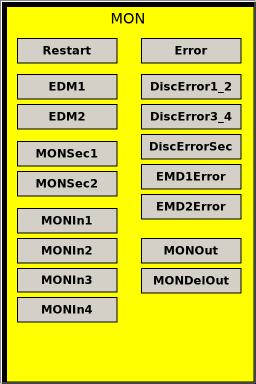
VISUALIZATION V_PH_MON  // 256x384
VAR_INPUT
	stSafetyMon				: ST_SAFETY_FBMON;
	
END_VAR
    Rectangle (2,2 256x384), colour toggle: stSafetyMon.bGeneralError
    Label (5,6 246x25), "MON"
    RoundedRectangle (17,38 100x25), "Restart", colour toggle: stSafetyMon.uStatus.stStatusWords.wInputs.0
    RoundedRectangle (17,74 100x25), "EDM1", colour toggle: stSafetyMon.uStatus.stStatusWords.wInputs.1
    RoundedRectangle (17,297 100x25), "MONIn4", colour toggle: stSafetyMon.uStatus.stStatusWords.wInputs.11
    RoundedRectangle (17,104 100x25), "EDM2", colour toggle: stSafetyMon.uStatus.stStatusWords.wInputs.2
    RoundedRectangle (17,171 100x25), "MONSec2", colour toggle: stSafetyMon.uStatus.stStatusWords.wInputs.4
    RoundedRectangle (17,268 100x24), "MONIn3", colour toggle: stSafetyMon.uStatus.stStatusWords.wInputs.10
    RoundedRectangle (17,141 100x25), "MONSec1", colour toggle: stSafetyMon.uStatus.stStatusWords.wInputs.3
    RoundedRectangle (17,238 100x25), "MONIn2", colour toggle: stSafetyMon.uStatus.stStatusWords.wInputs.9
    RoundedRectangle (17,208 100x25), "MONIn1", colour toggle: stSafetyMon.uStatus.stStatusWords.wInputs.8
    RoundedRectangle (141,74 100x25), "DiscError1_2", colour toggle: stSafetyMon.uStatus.stStatusWords.wDiagnosis.0, invisible if: NOT stSafetyMon.uStatus.stStatusWords.wDiagnosis.0
    RoundedRectangle (141,104 100x25), "DiscError3_4", colour toggle: stSafetyMon.uStatus.stStatusWords.wDiagnosis.1, invisible if: NOT stSafetyMon.uStatus.stStatusWords.wDiagnosis.1
    RoundedRectangle (141,134 100x25), "DiscErrorSec", colour toggle: stSafetyMon.uStatus.stStatusWords.wDiagnosis.2, invisible if: NOT stSafetyMon.uStatus.stStatusWords.wDiagnosis.2
    RoundedRectangle (141,194 100x25), "EMD2Error", colour toggle: stSafetyMon.uStatus.stStatusWords.wDiagnosis.5, invisible if: NOT stSafetyMon.uStatus.stStatusWords.wDiagnosis.5
    RoundedRectangle (141,164 100x25), "EMD1Error", colour toggle: stSafetyMon.uStatus.stStatusWords.wDiagnosis.4, invisible if: NOT stSafetyMon.uStatus.stStatusWords.wDiagnosis.4
    RoundedRectangle (141,38 100x25), "Error", colour toggle: stSafetyMon.uStatus.stStatusWords.wOutputs.0
    RoundedRectangle (141,238 100x25), "MONOut", colour toggle: stSafetyMon.uStatus.stStatusWords.wOutputs.1
    RoundedRectangle (141,268 100x25), "MONDelOut", colour toggle: stSafetyMon.uStatus.stStatusWords.wOutputs.2
    Textfield (17,354 234x25), text list: 'TL_FbState', text index: stSafetyMon.eState
END_VISUALIZATION

// ---- VISUs/FBs/V_PH_MUTING.TcVIS
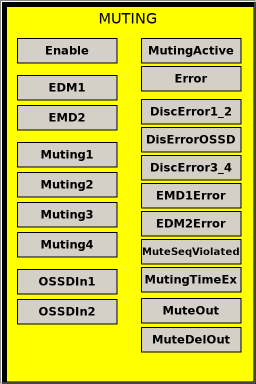
VISUALIZATION V_PH_MUTING  // 256x384
VAR_INPUT
	stSafetyMuting				:ST_SAFETY_FBMUTING;
END_VAR
    Rectangle (2,2 256x384), colour toggle: stSafetyMuting.bGeneralError
    RoundedRectangle (17,142 100x25), "Muting1", colour toggle: stSafetyMuting.uStatus.stStatusWords.wInputs.8
    RoundedRectangle (17,38 100x25), "Enable", colour toggle: stSafetyMuting.uStatus.stStatusWords.wInputs.0
    RoundedRectangle (17,105 100x25), "EMD2", colour toggle: stSafetyMuting.uStatus.stStatusWords.wInputs.2
    RoundedRectangle (17,172 100x25), "Muting2", colour toggle: stSafetyMuting.uStatus.stStatusWords.wInputs.9
    RoundedRectangle (17,202 100x25), "Muting3", colour toggle: stSafetyMuting.uStatus.stStatusWords.wInputs.10
    RoundedRectangle (17,299 100x25), "OSSDIn2", colour toggle: stSafetyMuting.uStatus.stStatusWords.wInputs.13
    RoundedRectangle (17,232 100x25), "Muting4", colour toggle: stSafetyMuting.uStatus.stStatusWords.wInputs.11
    RoundedRectangle (17,269 100x25), "OSSDIn1", colour toggle: stSafetyMuting.uStatus.stStatusWords.wInputs.12
    RoundedRectangle (17,75 100x25), "EDM1", colour toggle: stSafetyMuting.uStatus.stStatusWords.wInputs.1
    Label (5,6 246x25), "MUTING"
    RoundedRectangle (141,38 100x25), "MutingActive", colour toggle: stSafetyMuting.uStatus.stStatusWords.wOutputs.1
    RoundedRectangle (141,66 100x25), "Error", colour toggle: stSafetyMuting.uStatus.stStatusWords.wOutputs.0
    RoundedRectangle (141,298 100x25), "MuteOut", colour toggle: stSafetyMuting.uStatus.stStatusWords.wOutputs.2
    RoundedRectangle (141,327 100x25), "MuteDelOut", colour toggle: stSafetyMuting.uStatus.stStatusWords.wOutputs.3
    RoundedRectangle (141,127 100x25), "DisErrorOSSD", colour toggle: stSafetyMuting.uStatus.stStatusWords.wDiagnosis.1, invisible if: NOT stSafetyMuting.uStatus.stStatusWords.wDiagnosis.1
    RoundedRectangle (141,183 100x25), "EMD1Error", colour toggle: stSafetyMuting.uStatus.stStatusWords.wDiagnosis.4, invisible if: NOT stSafetyMuting.uStatus.stStatusWords.wDiagnosis.4
    RoundedRectangle (141,99 100x25), "DiscError1_2", colour toggle: stSafetyMuting.uStatus.stStatusWords.wDiagnosis.0, invisible if: NOT stSafetyMuting.uStatus.stStatusWords.wDiagnosis.0
    RoundedRectangle (141,155 100x25), "DiscError3_4", colour toggle: stSafetyMuting.uStatus.stStatusWords.wDiagnosis.2, invisible if: NOT stSafetyMuting.uStatus.stStatusWords.wDiagnosis.2
    RoundedRectangle (141,267 100x25), "MutingTimeEx", colour toggle: stSafetyMuting.uStatus.stStatusWords.wDiagnosis.7, invisible if: NOT stSafetyMuting.uStatus.stStatusWords.wDiagnosis.7
    RoundedRectangle (141,211 100x25), "EDM2Error", colour toggle: stSafetyMuting.uStatus.stStatusWords.wDiagnosis.5, invisible if: NOT stSafetyMuting.uStatus.stStatusWords.wDiagnosis.5
    RoundedRectangle (141,239 100x25), "MuteSeqViolated", colour toggle: stSafetyMuting.uStatus.stStatusWords.wDiagnosis.6, invisible if: NOT stSafetyMuting.uStatus.stStatusWords.wDiagnosis.6
    Textfield (17,354 234x25), text list: 'TL_FbStateMUTING', text index: stSafetyMuting.eState
END_VISUALIZATION

// ---- VISUs/FBs/V_PH_OPMODE.TcVIS
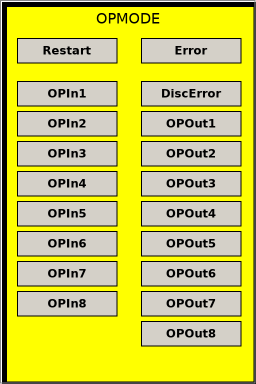
VISUALIZATION V_PH_OPMODE  // 256x384
VAR_INPUT
	stSafetyOPMODE			:ST_SAFETY_FBOPMODE;
END_VAR
    Rectangle (2,2 256x384), colour toggle: stSafetyOPMODE.bGeneralError
    Label (5,6 246x25), "OPMODE"
    RoundedRectangle (17,38 100x25), "Restart", colour toggle: stSafetyOPMODE.uStatus.stStatusWords.wInputs.0
    RoundedRectangle (17,81 100x25), "OPIn1", colour toggle: stSafetyOPMODE.uStatus.stStatusWords.wInputs.8
    RoundedRectangle (17,111 100x25), "OPIn2", colour toggle: stSafetyOPMODE.uStatus.stStatusWords.wInputs.9
    RoundedRectangle (17,201 100x25), "OPIn5", colour toggle: stSafetyOPMODE.uStatus.stStatusWords.wInputs.12
    RoundedRectangle (17,171 100x25), "OPIn4", colour toggle: stSafetyOPMODE.uStatus.stStatusWords.wInputs.11
    RoundedRectangle (17,141 100x25), "OPIn3", colour toggle: stSafetyOPMODE.uStatus.stStatusWords.wInputs.10
    RoundedRectangle (17,261 100x25), "OPIn7", colour toggle: stSafetyOPMODE.uStatus.stStatusWords.wInputs.14
    RoundedRectangle (17,291 100x25), "OPIn8", colour toggle: stSafetyOPMODE.uStatus.stStatusWords.wInputs.15
    RoundedRectangle (17,231 100x25), "OPIn6", colour toggle: stSafetyOPMODE.uStatus.stStatusWords.wInputs.13
    RoundedRectangle (141,81 100x25), "DiscError", colour toggle: stSafetyOPMODE.uStatus.stStatusWords.wDiagnosis.0, invisible if: NOT stSafetyOPMODE.uStatus.stStatusWords.wDiagnosis.0
    RoundedRectangle (141,38 100x25), "Error", colour toggle: stSafetyOPMODE.uStatus.stStatusWords.wOutputs.0
    RoundedRectangle (141,141 100x25), "OPOut2", colour toggle: stSafetyOPMODE.uStatus.stStatusWords.wOutputs.9
    RoundedRectangle (141,171 100x25), "OPOut3", colour toggle: stSafetyOPMODE.uStatus.stStatusWords.wOutputs.10
    RoundedRectangle (141,111 100x25), "OPOut1", colour toggle: stSafetyOPMODE.uStatus.stStatusWords.wOutputs.8
    RoundedRectangle (141,201 100x25), "OPOut4", colour toggle: stSafetyOPMODE.uStatus.stStatusWords.wOutputs.11
    RoundedRectangle (141,261 100x25), "OPOut6", colour toggle: stSafetyOPMODE.uStatus.stStatusWords.wOutputs.13
    RoundedRectangle (141,321 100x25), "OPOut8", colour toggle: stSafetyOPMODE.uStatus.stStatusWords.wOutputs.15
    RoundedRectangle (141,231 100x25), "OPOut5", colour toggle: stSafetyOPMODE.uStatus.stStatusWords.wOutputs.12
    RoundedRectangle (141,291 100x25), "OPOut7", colour toggle: stSafetyOPMODE.uStatus.stStatusWords.wOutputs.14
    Textfield (17,354 234x25), text list: 'TL_FbState', text index: stSafetyOPMODE.eState
END_VISUALIZATION

// ---- VISUs/FBs/V_PH_OR.TcVIS
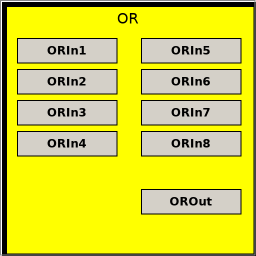
VISUALIZATION V_PH_OR  // 256x256
VAR_INPUT
	stSafetyOR			:ST_SAFETY_FBOR;
	
END_VAR
    Rectangle (2,2 256x256), colour toggle: stSafetyOR.bGeneralError
    Label (5,6 246x25), "OR"
    RoundedRectangle (17,38 100x25), "ORIn1", colour toggle: stSafetyOR.uStatus.stStatusWords.wInputs.8
    RoundedRectangle (17,100 100x25), "ORIn3", colour toggle: stSafetyOR.uStatus.stStatusWords.wInputs.10
    RoundedRectangle (17,131 100x25), "ORIn4", colour toggle: stSafetyOR.uStatus.stStatusWords.wInputs.11
    RoundedRectangle (141,38 100x25), "ORIn5", colour toggle: stSafetyOR.uStatus.stStatusWords.wInputs.12
    RoundedRectangle (141,69 100x25), "ORIn6", colour toggle: stSafetyOR.uStatus.stStatusWords.wInputs.13
    RoundedRectangle (141,100 100x25), "ORIn7", colour toggle: stSafetyOR.uStatus.stStatusWords.wInputs.14
    RoundedRectangle (141,131 100x25), "ORIn8", colour toggle: stSafetyOR.uStatus.stStatusWords.wInputs.15
    RoundedRectangle (17,69 100x25), "ORIn2", colour toggle: stSafetyOR.uStatus.stStatusWords.wInputs.9
    RoundedRectangle (141,189 100x25), "OROut", colour toggle: stSafetyOR.uStatus.stStatusWords.wOutputs.0
    Textfield (17,226 234x25), text list: 'TL_FbState', text index: stSafetyOR.eState
END_VISUALIZATION

// ---- VISUs/FBs/V_PH_RS.TcVIS
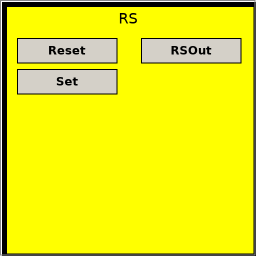
VISUALIZATION V_PH_RS  // 256x256
VAR_INPUT
	
	stSafetyRS				:ST_SAFETY_FBRS;
END_VAR
    Rectangle (2,2 256x256), colour toggle: stSafetyRS.bGeneralError
    Label (5,6 246x25), "RS"
    RoundedRectangle (17,38 100x25), "Reset", colour toggle: stSafetyRS.uStatus.stStatusWords.wInputs.8
    RoundedRectangle (141,38 100x25), "RSOut", colour toggle: stSafetyRS.uStatus.stStatusWords.wOutputs.1
    RoundedRectangle (17,69 100x25), "Set", colour toggle: stSafetyRS.uStatus.stStatusWords.wInputs.9
    Textfield (17,226 234x25), text list: 'TL_FbStateSetReset', text index: stSafetyRS.eState
END_VISUALIZATION

// ---- VISUs/FBs/V_PH_SR.TcVIS
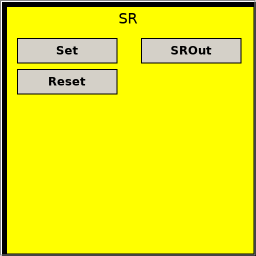
VISUALIZATION V_PH_SR  // 256x256
VAR_INPUT
	stSafetySR				:ST_SAFETY_FBSR;
END_VAR
    Rectangle (2,2 256x256), colour toggle: stSafetySR.bGeneralError
    Label (5,6 246x25), "SR"
    RoundedRectangle (17,69 100x25), "Reset", colour toggle: stSafetySR.uStatus.stStatusWords.wInputs.9
    RoundedRectangle (141,38 100x25), "SROut", colour toggle: stSafetySR.uStatus.stStatusWords.wOutputs.1
    RoundedRectangle (17,38 100x25), "Set", colour toggle: stSafetySR.uStatus.stStatusWords.wInputs.8
    Textfield (17,226 234x25), text list: 'TL_FbStateSetReset', text index: stSafetySR.eState
END_VISUALIZATION

// ---- VISUs/FBs/V_PH_TOF.TcVIS
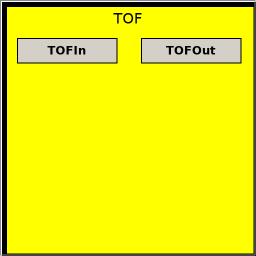
VISUALIZATION V_PH_TOF  // 256x256
VAR_INPUT
	stSafetyTOF			:ST_SAFETY_FBTOF;
END_VAR
    Rectangle (2,2 256x256), colour toggle: stSafetyTOF.bGeneralError
    Label (5,6 246x25), "TOF"
    RoundedRectangle (17,38 100x25), "TOFIn", colour toggle: stSafetyTOF.uStatus.stStatusWords.wInputs.8
    RoundedRectangle (141,38 100x25), "TOFOut", colour toggle: stSafetyTOF.uStatus.stStatusWords.wOutputs.1
    Textfield (17,226 234x25), text list: 'TL_FbStateTimer', text index: stSafetyTOF.eState
END_VISUALIZATION

// ---- VISUs/FBs/V_PH_TON.TcVIS
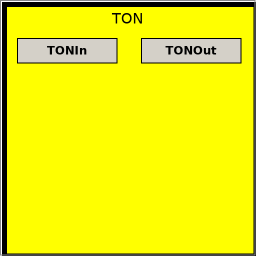
VISUALIZATION V_PH_TON  // 256x256
VAR_INPUT
	stSafetyTON			:ST_SAFETY_FBTON;
END_VAR
    Rectangle (2,2 256x256), colour toggle: stSafetyTON.bGeneralError
    Label (5,6 246x25), "TON"
    RoundedRectangle (17,38 100x25), "TONIn", colour toggle: stSafetyTON.uStatus.stStatusWords.wInputs.8
    RoundedRectangle (141,38 100x25), "TONOut", colour toggle: stSafetyTON.uStatus.stStatusWords.wOutputs.1
    Textfield (17,226 234x25), text list: 'TL_FbStateTimer', text index: stSafetyTON.eState
END_VISUALIZATION

// ---- VISUs/FBs/V_PH_TWOHAND.TcVIS
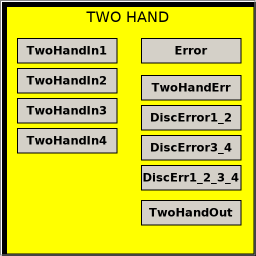
VISUALIZATION V_PH_TWOHAND  // 256x256
VAR_INPUT
	stSafetyTWOHAND			:ST_SAFETY_FBTWOHAND;
END_VAR
    Rectangle (2,2 256x256), colour toggle: stSafetyTWOHAND.bGeneralError
    Label (5,6 246x22), "TWO HAND"
    RoundedRectangle (17,38 100x25), "TwoHandIn1", colour toggle: stSafetyTWOHAND.uStatus.stStatusWords.wInputs.8
    RoundedRectangle (17,98 100x25), "TwoHandIn3", colour toggle: stSafetyTWOHAND.uStatus.stStatusWords.wInputs.10
    RoundedRectangle (17,68 100x25), "TwoHandIn2", colour toggle: stSafetyTWOHAND.uStatus.stStatusWords.wInputs.9
    RoundedRectangle (17,128 100x25), "TwoHandIn4", colour toggle: stSafetyTWOHAND.uStatus.stStatusWords.wInputs.11
    RoundedRectangle (141,38 100x25), "Error", colour toggle: stSafetyTWOHAND.uStatus.stStatusWords.wOutputs.0
    RoundedRectangle (141,200 100x25), "TwoHandOut", colour toggle: stSafetyTWOHAND.uStatus.stStatusWords.wOutputs.1
    RoundedRectangle (141,105 100x25), "DiscError1_2", colour toggle: stSafetyTWOHAND.uStatus.stStatusWords.wDiagnosis.0, invisible if: NOT stSafetyTWOHAND.uStatus.stStatusWords.wDiagnosis.0
    RoundedRectangle (141,75 100x25), "TwoHandErr", colour toggle: stSafetyTWOHAND.uStatus.stStatusWords.wDiagnosis.6
    RoundedRectangle (141,165 100x25), "DiscErr1_2_3_4", colour toggle: stSafetyTWOHAND.uStatus.stStatusWords.wDiagnosis.2, invisible if: NOT stSafetyTWOHAND.uStatus.stStatusWords.wDiagnosis.2
    RoundedRectangle (141,135 100x25), "DiscError3_4", colour toggle: stSafetyTWOHAND.uStatus.stStatusWords.wDiagnosis.1, invisible if: NOT stSafetyTWOHAND.uStatus.stStatusWords.wDiagnosis.1
    Textfield (17,226 234x25), text list: 'TL_FbState', text index: stSafetyTWOHAND.eState
END_VISUALIZATION

// ---- VISUs/HW/V_PH_EL1904_DIAG.TcVIS
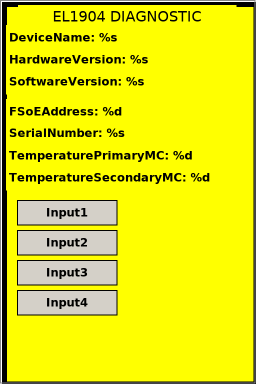
VISUALIZATION V_PH_EL1904_DIAG  // 256x384
VAR_INPUT
	stEL1904DiagnosticData		:ST_EL1904_DiagnosticData;
	
	
END_VAR
    Rectangle (2,2 256x384), colour toggle: stEL1904DiagnosticData.bGeneralError
    Rectangle (18,5 218x23), "EL1904 DIAGNOSTIC"
    Rectangle (6,25 242x25), "DeviceName: %s", text variable: stEL1904DiagnosticData.sDeviceName
    Rectangle (6,69 243x25), "SoftwareVersion: %s", text variable: stEL1904DiagnosticData.sSoftwareVersion
    Rectangle (6,47 243x25), "HardwareVersion: %s", text variable: stEL1904DiagnosticData.sHardwareVersion
    Rectangle (6,99 243x25), "FSoEAddress: %d", text variable: stEL1904DiagnosticData.dwFSoEAddress
    Rectangle (6,121 243x24), "SerialNumber: %s", text variable: stEL1904DiagnosticData.sSerialNumber
    Rectangle (6,165 243x25), "TemperatureSecondaryMC: %d", text variable: stEL1904DiagnosticData.wTemperatureSecondaryMC
    Rectangle (6,143 243x25), "TemperaturePrimaryMC: %d", text variable: stEL1904DiagnosticData.wTemperaturePrimaryMC
    RoundedRectangle (17,260 100x25), "Input3", colour toggle: stEL1904DiagnosticData.bInput3
    RoundedRectangle (17,290 100x25), "Input4", colour toggle: stEL1904DiagnosticData.bInput4
    RoundedRectangle (17,230 100x25), "Input2", colour toggle: stEL1904DiagnosticData.bInput2
    RoundedRectangle (17,200 100x25), "Input1", colour toggle: stEL1904DiagnosticData.bInput1
END_VISUALIZATION

// ---- VISUs/HW/V_PH_EL2904_DIAG.TcVIS
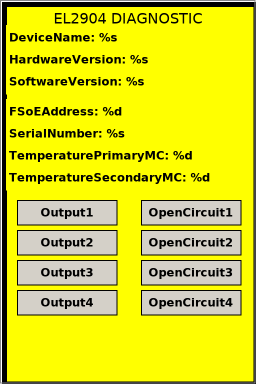
VISUALIZATION V_PH_EL2904_DIAG  // 256x384
VAR_INPUT
	stEL2904DiagnosticData		:ST_EL2904_DiagnosticData;
END_VAR
    Rectangle (2,2 256x384), colour toggle: stEL2904DiagnosticData.bGeneralError
    Label (5,6 246x25), "EL2904 DIAGNOSTIC"
    Rectangle (6,25 242x25), "DeviceName: %s", text variable: stEL2904DiagnosticData.sDeviceName
    Rectangle (6,47 242x25), "HardwareVersion: %s", text variable: stEL2904DiagnosticData.sHardwareVersion
    Rectangle (6,69 242x25), "SoftwareVersion: %s", text variable: stEL2904DiagnosticData.sSoftwareVersion
    Rectangle (6,99 242x25), "FSoEAddress: %d", text variable: stEL2904DiagnosticData.dwFSoEAddress
    Rectangle (6,121 242x25), "SerialNumber: %s", text variable: stEL2904DiagnosticData.sSerialNumber
    Rectangle (6,143 242x25), "TemperaturePrimaryMC: %d", text variable: stEL2904DiagnosticData.wTemperaturePrimaryMC
    Rectangle (6,165 242x25), "TemperatureSecondaryMC: %d", text variable: stEL2904DiagnosticData.wTemperatureSecondaryMC
    RoundedRectangle (17,200 100x25), "Output1", colour toggle: stEL2904DiagnosticData.bOutput1
    RoundedRectangle (17,230 100x25), "Output2", colour toggle: stEL2904DiagnosticData.bOutput2
    RoundedRectangle (17,260 100x25), "Output3", colour toggle: stEL2904DiagnosticData.bOutput3
    RoundedRectangle (17,290 100x25), "Output4", colour toggle: stEL2904DiagnosticData.bOutput4
    RoundedRectangle (141,200 100x25), "OpenCircuit1", colour toggle: stEL2904DiagnosticData.bOutputOpen1, invisible if: NOT stEL2904DiagnosticData.bOutputOpen1
    RoundedRectangle (141,230 100x25), "OpenCircuit2", colour toggle: stEL2904DiagnosticData.bOutputOpen2, invisible if: NOT stEL2904DiagnosticData.bOutputOpen2
    RoundedRectangle (141,260 100x25), "OpenCircuit3", colour toggle: stEL2904DiagnosticData.bOutputOpen3, invisible if: NOT stEL2904DiagnosticData.bOutputOpen3
    RoundedRectangle (141,290 100x25), "OpenCircuit4", colour toggle: stEL2904DiagnosticData.bOutputOpen4, invisible if: NOT stEL2904DiagnosticData.bOutputOpen4
END_VISUALIZATION

// ---- VISUs/HW/V_PH_EL6900_DIAG.TcVIS
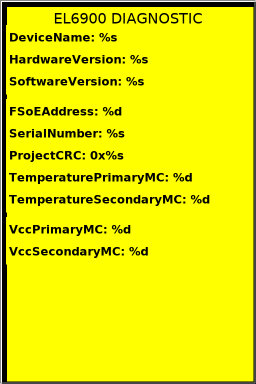
VISUALIZATION V_PH_EL6900_DIAG  // 256x384
VAR_INPUT
	stEL6900DiagnosticData		:ST_EL6900_DiagnosticData;
END_VAR
    Rectangle (2,2 256x384), colour toggle: stEL6900DiagnosticData.bGeneralError
    Label (5,6 246x25), "EL6900 DIAGNOSTIC"
    Rectangle (6,25 242x25), "DeviceName: %s", text variable: stEL6900DiagnosticData.sDeviceName
    Rectangle (6,47 242x25), "HardwareVersion: %s", text variable: stEL6900DiagnosticData.sHardwareVersion
    Rectangle (6,69 242x25), "SoftwareVersion: %s", text variable: stEL6900DiagnosticData.sSoftwareVersion
    Rectangle (6,121 242x25), "SerialNumber: %s", text variable: stEL6900DiagnosticData.sSerialNumber
    Rectangle (6,143 242x25), "ProjectCRC: 0x%s", text variable: stEL6900DiagnosticData.sProjectCRC
    Rectangle (6,187 242x25), "TemperatureSecondaryMC: %d", text variable: stEL6900DiagnosticData.wTemperatureSecondaryMC
    Rectangle (6,99 242x25), "FSoEAddress: %d", text variable: stEL6900DiagnosticData.dwFSoEAddress
    Rectangle (6,165 242x25), "TemperaturePrimaryMC: %d", text variable: stEL6900DiagnosticData.wTemperaturePrimaryMC
    Rectangle (6,217 242x25), "VccPrimaryMC: %d", text variable: stEL6900DiagnosticData.wVccPrimaryMC
    Rectangle (6,239 242x25), "VccSecondaryMC: %d", text variable: stEL6900DiagnosticData.wVccSecondaryMC
END_VISUALIZATION

// ---- VISUs/V_PH_CONNECTION.TcVIS
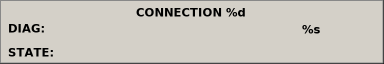
VISUALIZATION V_PH_CONNECTION  // 384x64
VAR_INPUT
		wIndex						: WORD;
		stSafetyStausConnection		:ST_SAFETYStatusConnection;
END_VAR
    Rectangle (0,0 384x64)
    Rectangle (102,1 178x23), "CONNECTION %d", text variable: wIndex
    Rectangle (60,17 232x25), text list: 'TL_ConnectionDiag', text index: stSafetyStausConnection.eSAFETY_ConnectionDiag0F
    Rectangle (299,17 75x25), "%s", text variable: stSafetyStausConnection.sSAFETY_ConnectionDiagF0
    Rectangle (60,38 314x25), text list: 'TL_ConnectionState', text index: stSafetyStausConnection.eSAFETY_ConnectionState
    Label (5,18 43x21), "DIAG:"
    Label (5,38 51x29), "STATE:"
END_VISUALIZATION

// ---- VISUs/V_PH_GROUP.TcVIS
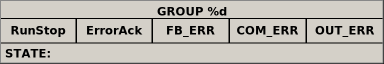
VISUALIZATION V_PH_GROUP  // 384x64
VAR_INPUT
	wIndex					:WORD;
	stSafetyStatusGroup		:ST_SAFETYStatusGroup;
	
END_VAR
    Rectangle (0,0 384x64)
    Rectangle (117,1 150x21), "GROUP %d", text variable: wIndex
    Rectangle (76,18 76x25), "ErrorAck", colour toggle: stSafetyStatusGroup.bERR_Ack
    Rectangle (152,18 77x25), "FB_ERR", colour toggle: stSafetyStatusGroup.bFB_ERR
    Rectangle (306,18 78x25), "OUT_ERR", colour toggle: stSafetyStatusGroup.bOUT_ERR
    Rectangle (229,18 77x25), "COM_ERR", colour toggle: stSafetyStatusGroup.bCOM_ERR
    Rectangle (0,18 76x25), "RunStop", colour toggle: stSafetyStatusGroup.bRUN_STOP
    Rectangle (67,44 315x19), text list: 'TL_GroupState', text index: stSafetyStatusGroup.eSAFETY_GroupState
    Label (2,44 55x19), "STATE:"
END_VISUALIZATION
